LIN {X 0,Y 532.098,Z 319.802,A -85,B 0,C 180,E1 -4422.927,E2 -4422.927} C_VEL
LIN {X 0,Y 532.084,Z 308.331,A -85,B 0,C 180,E1 -4423.281,E2 -4423.281} C_VEL
LIN {X 0,Y 530.627,Z 298.644,A -85,B 0,C 180,E1 -4423.524,E2 -4423.524} C_VEL
LIN {X 0,Y 530.739,Z 289.457,A -85,B 0,C 180,E1 -4426.146,E2 -4426.146} C_VEL
LIN {X 0,Y 530.824,Z 279.726,A -85,B 0,C 180,E1 -4428.928,E2 -4428.928} C_VEL
LIN {X 0,Y 530.984,Z 268.988,A -85,B 0,C 180,E1 -4432.103,E2 -4432.103} C_VEL
LIN {X 0,Y 531.056,Z 259.338,A -85,B 0,C 180,E1 -4435.055,E2 -4435.055} C_VEL
LIN {X 0,Y 531.227,Z 250.169,A -85,B 0,C 180,E1 -4438.012,E2 -4438.012} C_VEL
LIN {X 0,Y 531.545,Z 241.433,A -85,B 0,C 180,E1 -4441.041,E2 -4441.041} C_VEL
LIN {X 0,Y 532.022,Z 233.376,A -85,B 0,C 180,E1 -4444.155,E2 -4444.155} C_VEL
LIN {X 0,Y 532.107,Z 230.247,A -85,B 0,C 180,E1 -4445.532,E2 -4445.532} C_VEL
LIN {X 0,Y 531.699,Z 226.333,A -85,B 0,C 180,E1 -4447.526,E2 -4447.526} C_VEL
LIN {X 0,Y 531.191,Z 223.293,A -85,B 0,C 180,E1 -4449.426,E2 -4449.426} C_VEL
LIN {X 0,Y 530.987,Z 222.375,A -85,B 0,C 180,E1 -4450.111,E2 -4450.111} C_VEL
LIN {X 0,Y 530.981,Z 222.346,A -85,B 0,C 180,E1 -4452.457,E2 -4452.457} C_VEL
LIN {X 0,Y 530.981,Z 222.348,A -85,B 0,C 180,E1 -4455.622,E2 -4455.622} C_VEL
LIN {X 0,Y 530.997,Z 222.344,A -85,B 0,C 180,E1 -4458.565,E2 -4458.565} C_VEL
LIN {X 0,Y 530.962,Z 222.35,A -85,B 0,C 180,E1 -4461.53,E2 -4461.53} C_VEL
LIN {X 0,Y 530.954,Z 222.351,A -85,B 0,C 180,E1 -4464.38,E2 -4464.38} C_VEL
LIN {X 0,Y 530.987,Z 222.799,A -85,B 0,C 180,E1 -4465.31,E2 -4465.31} C_VEL
LIN {X 0,Y 530.925,Z 225.158,A -85,B 0,C 180,E1 -4468.029,E2 -4468.029} C_VEL
LIN {X 0,Y 530.845,Z 227.83,A -85,B 0,C 180,E1 -4470.903,E2 -4470.903} C_VEL
LIN {X 0,Y 530.76,Z 231.038,A -85,B 0,C 180,E1 -4474.213,E2 -4474.213} C_VEL
LIN {X 0,Y 530.662,Z 233.419,A -85,B 0,C 180,E1 -4476.59,E2 -4476.59} C_VEL
LIN {X 0,Y 530.617,Z 235.93,A -85,B 0,C 180,E1 -4479.046,E2 -4479.046} C_VEL
LIN {X 0,Y 530.598,Z 239.55,A -85,B 0,C 180,E1 -4482.493,E2 -4482.493} C_VEL
LIN {X 0,Y 530.553,Z 242.668,A -85,B 0,C 180,E1 -4485.423,E2 -4485.423} C_VEL
LIN {X 0,Y 530.522,Z 245.123,A -85,B 0,C 180,E1 -4487.605,E2 -4487.605} C_VEL
LIN {X 0,Y 532.268,Z 254.517,A -85,B 0,C 180,E1 -4487.886,E2 -4487.886} C_VEL
LIN {X 0,Y 532.14,Z 267.138,A -85,B 0,C 180,E1 -4488.336,E2 -4488.336} C_VEL
LIN {X 0,Y 531.892,Z 278.037,A -85,B 0,C 180,E1 -4488.858,E2 -4488.858} C_VEL
LIN {X 0,Y 531.608,Z 288.977,A -85,B 0,C 180,E1 -4489.527,E2 -4489.527} C_VEL
LIN {X 0,Y 531.384,Z 300.143,A -85,B 0,C 180,E1 -4490.388,E2 -4490.388} C_VEL
LIN {X 0,Y 531.175,Z 309.139,A -85,B 0,C 180,E1 -4491.248,E2 -4491.248} C_VEL
LIN {X 0,Y 530.932,Z 317.38,A -85,B 0,C 180,E1 -4492.202,E2 -4492.202} C_VEL
LIN {X 0,Y 530.778,Z 324.845,A -85,B 0,C 180,E1 -4493.255,E2 -4493.255} C_VEL
LIN {X 0,Y 530.663,Z 330.911,A -85,B 0,C 180,E1 -4494.3,E2 -4494.3} C_VEL
LIN {X 0,Y 530.602,Z 336.255,A -85,B 0,C 180,E1 -4495.442,E2 -4495.442} C_VEL
LIN {X 0,Y 530.567,Z 340.431,A -85,B 0,C 180,E1 -4496.583,E2 -4496.583} C_VEL
LIN {X 0,Y 530.431,Z 343.565,A -85,B 0,C 180,E1 -4497.722,E2 -4497.722} C_VEL
LIN {X 0,Y 530.373,Z 345.123,A -85,B 0,C 180,E1 -4498.481,E2 -4498.481} C_VEL
LIN {X 0,Y 530.355,Z 346.27,A -85,B 0,C 180,E1 -4499.241,E2 -4499.241} C_VEL
LIN {X 0,Y 530.351,Z 347.32,A -85,B 0,C 180,E1 -4500.759,E2 -4500.759} C_VEL
LIN {X 0,Y 530.411,Z 346.844,A -85,B 0,C 180,E1 -4502.278,E2 -4502.278} C_VEL
LIN {X 0,Y 530.482,Z 345.982,A -85,B 0,C 180,E1 -4503.038,E2 -4503.038} C_VEL
LIN {X 0,Y 530.489,Z 344.731,A -85,B 0,C 180,E1 -4503.798,E2 -4503.798} C_VEL
LIN {X 0,Y 530.441,Z 342.081,A -85,B 0,C 180,E1 -4504.941,E2 -4504.941} C_VEL
LIN {X 0,Y 530.554,Z 338.414,A -85,B 0,C 180,E1 -4506.083,E2 -4506.083} C_VEL
LIN {X 0,Y 530.61,Z 333.633,A -85,B 0,C 180,E1 -4507.229,E2 -4507.229} C_VEL
LIN {X 0,Y 530.755,Z 327.585,A -85,B 0,C 180,E1 -4508.375,E2 -4508.375} C_VEL
LIN {X 0,Y 530.878,Z 320.048,A -85,B 0,C 180,E1 -4509.525,E2 -4509.525} C_VEL
LIN {X 0,Y 531.079,Z 312.325,A -85,B 0,C 180,E1 -4510.484,E2 -4510.484} C_VEL
LIN {X 0,Y 531.333,Z 302.877,A -85,B 0,C 180,E1 -4511.444,E2 -4511.444} C_VEL
LIN {X 0,Y 531.503,Z 292.376,A -85,B 0,C 180,E1 -4512.311,E2 -4512.311} C_VEL
LIN {X 0,Y 531.862,Z 280.673,A -85,B 0,C 180,E1 -4513.079,E2 -4513.079} C_VEL
LIN {X 0,Y 532.065,Z 268.141,A -85,B 0,C 180,E1 -4513.706,E2 -4513.706} C_VEL
LIN {X 0,Y 532.272,Z 254.968,A -85,B 0,C 180,E1 -4514.188,E2 -4514.188} C_VEL
LIN {X 0,Y 530.472,Z 244.548,A -85,B 0,C 180,E1 -4514.506,E2 -4514.506} C_VEL
LIN {X 0,Y 530.488,Z 240.752,A -85,B 0,C 180,E1 -4517.741,E2 -4517.741} C_VEL
LIN {X 0,Y 530.476,Z 237.972,A -85,B 0,C 180,E1 -4520.149,E2 -4520.149} C_VEL
LIN {X 0,Y 530.473,Z 235.149,A -85,B 0,C 180,E1 -4522.595,E2 -4522.595} C_VEL
LIN {X 0,Y 530.536,Z 232.305,A -85,B 0,C 180,E1 -4525.081,E2 -4525.081} C_VEL
LIN {X 0,Y 530.579,Z 229.376,A -85,B 0,C 180,E1 -4527.62,E2 -4527.62} C_VEL
LIN {X 0,Y 530.596,Z 226.016,A -85,B 0,C 180,E1 -4530.575,E2 -4530.575} C_VEL
LIN {X 0,Y 530.623,Z 222.811,A -85,B 0,C 180,E1 -4533.443,E2 -4533.443} C_VEL
LIN {X 0,Y 530.64,Z 222.412,A -85,B 0,C 180,E1 -4533.798,E2 -4533.798} C_VEL
LIN {X 0,Y 530.907,Z 222.354,A -85,B 0,C 180,E1 -4536.563,E2 -4536.563} C_VEL
LIN {X 0,Y 530.94,Z 222.347,A -85,B 0,C 180,E1 -4538.185,E2 -4538.185} C_VEL
LIN {X 0,Y 530.31,Z 222.429,A -85,B 0,C 180,E1 -4538.819,E2 -4538.819} C_VEL
LIN {X 0,Y 527.489,Z 222.782,A -85,B 0,C 180,E1 -4539.847,E2 -4539.847} C_VEL
LIN {X 0,Y 525.079,Z 223.08,A -85,B 0,C 180,E1 -4540.674,E2 -4540.674} C_VEL
LIN {X 0,Y 524.034,Z 223.208,A -85,B 0,C 180,E1 -4541.314,E2 -4541.314} C_VEL
LIN {X 0,Y 523.944,Z 223.219,A -85,B 0,C 180,E1 -4541.53,E2 -4541.53} C_VEL
LIN {X 0,Y 523.945,Z 223.217,A -85,B 0,C 180,E1 -4544.689,E2 -4544.689} C_VEL
LIN {X 0,Y 523.912,Z 223.222,A -85,B 0,C 180,E1 -4547.877,E2 -4547.877} C_VEL
LIN {X 0,Y 523.903,Z 223.228,A -85,B 0,C 180,E1 -4550.913,E2 -4550.913} C_VEL
LIN {X 0,Y 523.858,Z 223.227,A -85,B 0,C 180,E1 -4553.821,E2 -4553.821} C_VEL
LIN {X 0,Y 523.916,Z 223.227,A -85,B 0,C 180,E1 -4556.633,E2 -4556.633} C_VEL
LIN {X 0,Y 523.948,Z 223.216,A -85,B 0,C 180,E1 -4559.355,E2 -4559.355} C_VEL
LIN {X 0,Y 523.951,Z 223.221,A -85,B 0,C 180,E1 -4562.288,E2 -4562.288} C_VEL
LIN {X 0,Y 523.932,Z 223.22,A -85,B 0,C 180,E1 -4564.58,E2 -4564.58} C_VEL
LIN {X 0,Y 523.915,Z 223.223,A -85,B 0,C 180,E1 -4567.106,E2 -4567.106} C_VEL
LIN {X 0,Y 523.984,Z 223.215,A -85,B 0,C 180,E1 -4569.866,E2 -4569.866} C_VEL
LIN {X 0,Y 523.955,Z 223.22,A -85,B 0,C 180,E1 -4572.837,E2 -4572.837} C_VEL
LIN {X 0,Y 523.978,Z 223.218,A -85,B 0,C 180,E1 -4575.236,E2 -4575.236} C_VEL
LIN {X 0,Y 524.018,Z 223.213,A -85,B 0,C 180,E1 -4578.394,E2 -4578.394} C_VEL
LIN {X 0,Y 523.957,Z 223.216,A -85,B 0,C 180,E1 -4581.515,E2 -4581.515} C_VEL
LIN {X 0,Y 524.028,Z 223.208,A -85,B 0,C 180,E1 -4584.613,E2 -4584.613} C_VEL
LIN {X 0,Y 524.106,Z 223.202,A -85,B 0,C 180,E1 -4587.694,E2 -4587.694} C_VEL
LIN {X 0,Y 524.104,Z 223.2,A -85,B 0,C 180,E1 -4590,E2 -4590} C_VEL
LIN {X 0,Y 524.043,Z 223.208,A -85,B 0,C 180,E1 -4593.075,E2 -4593.075} C_VEL
LIN {X 0,Y 523.728,Z 223.269,A -85,B 0,C 180,E1 -4595.728,E2 -4595.728} C_VEL
LIN {X 0,Y 523.74,Z 227.795,A -85,B 0,C 180,E1 -4597.712,E2 -4597.712} C_VEL
LIN {X 0,Y 523.7,Z 234.811,A -85,B 0,C 180,E1 -4600.829,E2 -4600.829} C_VEL
LIN {X 0,Y 523.643,Z 241.835,A -85,B 0,C 180,E1 -4603.98,E2 -4603.98} C_VEL
LIN {X 0,Y 523.592,Z 247.093,A -85,B 0,C 180,E1 -4606.372,E2 -4606.372} C_VEL
LIN {X 0,Y 523.568,Z 252.374,A -85,B 0,C 180,E1 -4608.793,E2 -4608.793} C_VEL
LIN {X 0,Y 523.481,Z 257.718,A -85,B 0,C 180,E1 -4611.253,E2 -4611.253} C_VEL
LIN {X 0,Y 523.449,Z 263.864,A -85,B 0,C 180,E1 -4614.077,E2 -4614.077} C_VEL
LIN {X 0,Y 523.466,Z 268.522,A -85,B 0,C 180,E1 -4616.266,E2 -4616.266} C_VEL
LIN {X 0,Y 524.612,Z 277.602,A -85,B 0,C 180,E1 -4616.558,E2 -4616.558} C_VEL
LIN {X 0,Y 524.443,Z 289.493,A -85,B 0,C 180,E1 -4617.052,E2 -4617.052} C_VEL
LIN {X 0,Y 524.275,Z 298.999,A -85,B 0,C 180,E1 -4617.602,E2 -4617.602} C_VEL
LIN {X 0,Y 524.117,Z 307.314,A -85,B 0,C 180,E1 -4618.208,E2 -4618.208} C_VEL
LIN {X 0,Y 523.983,Z 314.738,A -85,B 0,C 180,E1 -4618.872,E2 -4618.872} C_VEL
LIN {X 0,Y 523.833,Z 321.728,A -85,B 0,C 180,E1 -4619.631,E2 -4619.631} C_VEL
LIN {X 0,Y 523.656,Z 329.312,A -85,B 0,C 180,E1 -4620.664,E2 -4620.664} C_VEL
LIN {X 0,Y 523.583,Z 334.586,A -85,B 0,C 180,E1 -4621.567,E2 -4621.567} C_VEL
LIN {X 0,Y 523.433,Z 338.885,A -85,B 0,C 180,E1 -4622.484,E2 -4622.484} C_VEL
LIN {X 0,Y 523.417,Z 343.011,A -85,B 0,C 180,E1 -4623.645,E2 -4623.645} C_VEL
LIN {X 0,Y 523.316,Z 346.207,A -85,B 0,C 180,E1 -4624.993,E2 -4624.993} C_VEL
LIN {X 0,Y 523.293,Z 347.688,A -85,B 0,C 180,E1 -4626.31,E2 -4626.31} C_VEL
LIN {X 0,Y 523.248,Z 347.784,A -85,B 0,C 180,E1 -4627.584,E2 -4627.584} C_VEL
LIN {X 0,Y 523.269,Z 347.456,A -85,B 0,C 180,E1 -4628.158,E2 -4628.158} C_VEL
LIN {X 0,Y 523.312,Z 346.143,A -85,B 0,C 180,E1 -4629.139,E2 -4629.139} C_VEL
LIN {X 0,Y 523.389,Z 343.95,A -85,B 0,C 180,E1 -4630.131,E2 -4630.131} C_VEL
LIN {X 0,Y 523.435,Z 340.367,A -85,B 0,C 180,E1 -4631.245,E2 -4631.245} C_VEL
LIN {X 0,Y 523.516,Z 335.247,A -85,B 0,C 180,E1 -4632.408,E2 -4632.408} C_VEL
LIN {X 0,Y 523.624,Z 329.683,A -85,B 0,C 180,E1 -4633.378,E2 -4633.378} C_VEL
LIN {X 0,Y 523.771,Z 323.495,A -85,B 0,C 180,E1 -4634.246,E2 -4634.246} C_VEL
LIN {X 0,Y 523.966,Z 315.668,A -85,B 0,C 180,E1 -4635.132,E2 -4635.132} C_VEL
LIN {X 0,Y 524.107,Z 307.523,A -85,B 0,C 180,E1 -4635.871,E2 -4635.871} C_VEL
LIN {X 0,Y 524.296,Z 298.844,A -85,B 0,C 180,E1 -4636.504,E2 -4636.504} C_VEL
LIN {X 0,Y 524.511,Z 288.092,A -85,B 0,C 180,E1 -4637.111,E2 -4637.111} C_VEL
LIN {X 0,Y 524.614,Z 276.997,A -85,B 0,C 180,E1 -4637.554,E2 -4637.554} C_VEL
LIN {X 0,Y 523.439,Z 268.659,A -85,B 0,C 180,E1 -4637.83,E2 -4637.83} C_VEL
LIN {X 0,Y 523.494,Z 262.077,A -85,B 0,C 180,E1 -4640.877,E2 -4640.877} C_VEL
LIN {X 0,Y 523.487,Z 255.721,A -85,B 0,C 180,E1 -4643.792,E2 -4643.792} C_VEL
LIN {X 0,Y 523.611,Z 249.505,A -85,B 0,C 180,E1 -4646.611,E2 -4646.611} C_VEL
LIN {X 0,Y 523.578,Z 243.42,A -85,B 0,C 180,E1 -4649.331,E2 -4649.331} C_VEL
LIN {X 0,Y 523.635,Z 237.419,A -85,B 0,C 180,E1 -4651.981,E2 -4651.981} C_VEL
LIN {X 0,Y 523.641,Z 230.395,A -85,B 0,C 180,E1 -4654.99,E2 -4654.99} C_VEL
LIN {X 0,Y 523.728,Z 223.254,A -85,B 0,C 180,E1 -4657.982,E2 -4657.982} C_VEL
LIN {X 0,Y 523.963,Z 223.22,A -85,B 0,C 180,E1 -4660.407,E2 -4660.407} C_VEL
LIN {X 0,Y 523.958,Z 223.22,A -85,B 0,C 180,E1 -4662.837,E2 -4662.837} C_VEL
LIN {X 0,Y 523.979,Z 223.217,A -85,B 0,C 180,E1 -4665.236,E2 -4665.236} C_VEL
LIN {X 0,Y 524.016,Z 223.215,A -85,B 0,C 180,E1 -4668.394,E2 -4668.394} C_VEL
LIN {X 0,Y 524.007,Z 223.214,A -85,B 0,C 180,E1 -4671.516,E2 -4671.516} C_VEL
LIN {X 0,Y 524.075,Z 223.205,A -85,B 0,C 180,E1 -4674.613,E2 -4674.613} C_VEL
LIN {X 0,Y 524.115,Z 223.202,A -85,B 0,C 180,E1 -4677.694,E2 -4677.694} C_VEL
LIN {X 0,Y 524.124,Z 223.199,A -85,B 0,C 180,E1 -4680.768,E2 -4680.768} C_VEL
LIN {X 0,Y 524.072,Z 223.205,A -85,B 0,C 180,E1 -4683.075,E2 -4683.075} C_VEL
LIN {X 0,Y 524.029,Z 223.213,A -85,B 0,C 180,E1 -4686.159,E2 -4686.159} C_VEL
LIN {X 0,Y 524.004,Z 223.216,A -85,B 0,C 180,E1 -4688.484,E2 -4688.484} C_VEL
LIN {X 0,Y 524.007,Z 223.214,A -85,B 0,C 180,E1 -4691.739,E2 -4691.739} C_VEL
LIN {X 0,Y 523.997,Z 223.215,A -85,B 0,C 180,E1 -4695.052,E2 -4695.052} C_VEL
LIN {X 0,Y 523.95,Z 223.223,A -85,B 0,C 180,E1 -4697.969,E2 -4697.969} C_VEL
LIN {X 0,Y 523.975,Z 223.219,A -85,B 0,C 180,E1 -4700.41,E2 -4700.41} C_VEL
LIN {X 0,Y 523.914,Z 223.227,A -85,B 0,C 180,E1 -4702.893,E2 -4702.893} C_VEL
LIN {X 0,Y 523.946,Z 223.222,A -85,B 0,C 180,E1 -4706.01,E2 -4706.01} C_VEL
LIN {X 0,Y 523.937,Z 223.222,A -85,B 0,C 180,E1 -4708.875,E2 -4708.875} C_VEL
LIN {X 0,Y 523.922,Z 223.223,A -85,B 0,C 180,E1 -4711.544,E2 -4711.544} C_VEL
LIN {X 0,Y 523.923,Z 223.224,A -85,B 0,C 180,E1 -4714.291,E2 -4714.291} C_VEL
LIN {X 0,Y 523.91,Z 223.227,A -85,B 0,C 180,E1 -4717.132,E2 -4717.132} C_VEL
LIN {X 0,Y 523.94,Z 223.221,A -85,B 0,C 180,E1 -4720.13,E2 -4720.13} C_VEL
LIN {X 0,Y 523.937,Z 223.222,A -85,B 0,C 180,E1 -4722.459,E2 -4722.459} C_VEL
LIN {X 0,Y 523.946,Z 223.224,A -85,B 0,C 180,E1 -4725.31,E2 -4725.31} C_VEL
LIN {X 0,Y 523.958,Z 223.221,A -85,B 0,C 180,E1 -4728.69,E2 -4728.69} C_VEL
LIN {X 0,Y 523.954,Z 223.362,A -85,B 0,C 180,E1 -4731.595,E2 -4731.595} C_VEL
LIN {X 0,Y 524.95,Z 229.317,A -85,B 0,C 180,E1 -4733.909,E2 -4733.909} C_VEL
LIN {X 0,Y 524.989,Z 235.318,A -85,B 0,C 180,E1 -4736.098,E2 -4736.098} C_VEL
LIN {X 0,Y 524.695,Z 243.654,A -85,B 0,C 180,E1 -4739.009,E2 -4739.009} C_VEL
LIN {X 0,Y 524.336,Z 253.187,A -85,B 0,C 180,E1 -4742.207,E2 -4742.207} C_VEL
LIN {X 0,Y 524.169,Z 261.804,A -85,B 0,C 180,E1 -4745.017,E2 -4745.017} C_VEL
LIN {X 0,Y 523.984,Z 271.06,A -85,B 0,C 180,E1 -4747.941,E2 -4747.941} C_VEL
LIN {X 0,Y 523.837,Z 280.341,A -85,B 0,C 180,E1 -4750.81,E2 -4750.81} C_VEL
LIN {X 0,Y 523.672,Z 291.052,A -85,B 0,C 180,E1 -4754.031,E2 -4754.031} C_VEL
LIN {X 0,Y 523.592,Z 298.662,A -85,B 0,C 180,E1 -4756.291,E2 -4756.291} C_VEL
LIN {X 0,Y 525.346,Z 311.496,A -85,B 0,C 180,E1 -4756.633,E2 -4756.633} C_VEL
LIN {X 0,Y 525.105,Z 323.517,A -85,B 0,C 180,E1 -4757.045,E2 -4757.045} C_VEL
LIN {X 0,Y 524.816,Z 335.824,A -85,B 0,C 180,E1 -4757.628,E2 -4757.628} C_VEL
LIN {X 0,Y 524.526,Z 346.977,A -85,B 0,C 180,E1 -4758.31,E2 -4758.31} C_VEL
LIN {X 0,Y 524.308,Z 358.307,A -85,B 0,C 180,E1 -4759.184,E2 -4759.184} C_VEL
LIN {X 0,Y 524.003,Z 368.366,A -85,B 0,C 180,E1 -4760.154,E2 -4760.154} C_VEL
LIN {X 0,Y 523.776,Z 378.119,A -85,B 0,C 180,E1 -4761.318,E2 -4761.318} C_VEL
LIN {X 0,Y 523.612,Z 385.896,A -85,B 0,C 180,E1 -4762.48,E2 -4762.48} C_VEL
LIN {X 0,Y 523.482,Z 393.051,A -85,B 0,C 180,E1 -4763.834,E2 -4763.834} C_VEL
LIN {X 0,Y 523.383,Z 397.812,A -85,B 0,C 180,E1 -4764.993,E2 -4764.993} C_VEL
LIN {X 0,Y 523.443,Z 401.456,A -85,B 0,C 180,E1 -4766.151,E2 -4766.151} C_VEL
LIN {X 0,Y 523.367,Z 403.328,A -85,B 0,C 180,E1 -4766.921,E2 -4766.921} C_VEL
LIN {X 0,Y 523.335,Z 404.733,A -85,B 0,C 180,E1 -4767.691,E2 -4767.691} C_VEL
LIN {X 0,Y 523.254,Z 406.343,A -85,B 0,C 180,E1 -4769.231,E2 -4769.231} C_VEL
LIN {X 0,Y 523.254,Z 406.556,A -85,B 0,C 180,E1 -4770,E2 -4770} C_VEL
LIN {X 0,Y 523.275,Z 405.721,A -85,B 0,C 180,E1 -4771.539,E2 -4771.539} C_VEL
LIN {X 0,Y 523.335,Z 404.718,A -85,B 0,C 180,E1 -4772.309,E2 -4772.309} C_VEL
LIN {X 0,Y 523.367,Z 403.301,A -85,B 0,C 180,E1 -4773.079,E2 -4773.079} C_VEL
LIN {X 0,Y 523.424,Z 400.331,A -85,B 0,C 180,E1 -4774.235,E2 -4774.235} C_VEL
LIN {X 0,Y 523.461,Z 396.306,A -85,B 0,C 180,E1 -4775.393,E2 -4775.393} C_VEL
LIN {X 0,Y 523.515,Z 391.014,A -85,B 0,C 180,E1 -4776.574,E2 -4776.574} C_VEL
LIN {X 0,Y 523.649,Z 384.588,A -85,B 0,C 180,E1 -4777.713,E2 -4777.713} C_VEL
LIN {X 0,Y 523.821,Z 376.445,A -85,B 0,C 180,E1 -4778.876,E2 -4778.876} C_VEL
LIN {X 0,Y 523.992,Z 368.138,A -85,B 0,C 180,E1 -4779.847,E2 -4779.847} C_VEL
LIN {X 0,Y 524.267,Z 358.003,A -85,B 0,C 180,E1 -4780.817,E2 -4780.817} C_VEL
LIN {X 0,Y 524.475,Z 347.981,A -85,B 0,C 180,E1 -4781.596,E2 -4781.596} C_VEL
LIN {X 0,Y 524.734,Z 336.619,A -85,B 0,C 180,E1 -4782.304,E2 -4782.304} C_VEL
LIN {X 0,Y 525.055,Z 324.104,A -85,B 0,C 180,E1 -4782.907,E2 -4782.907} C_VEL
LIN {X 0,Y 525.275,Z 311.692,A -85,B 0,C 180,E1 -4783.344,E2 -4783.344} C_VEL
LIN {X 0,Y 523.553,Z 298.144,A -85,B 0,C 180,E1 -4783.71,E2 -4783.71} C_VEL
LIN {X 0,Y 523.67,Z 287.615,A -85,B 0,C 180,E1 -4786.771,E2 -4786.771} C_VEL
LIN {X 0,Y 523.757,Z 277.96,A -85,B 0,C 180,E1 -4789.601,E2 -4789.601} C_VEL
LIN {X 0,Y 523.908,Z 268.267,A -85,B 0,C 180,E1 -4792.527,E2 -4792.527} C_VEL
LIN {X 0,Y 524.023,Z 259.064,A -85,B 0,C 180,E1 -4795.415,E2 -4795.415} C_VEL
LIN {X 0,Y 524.202,Z 250.009,A -85,B 0,C 180,E1 -4798.422,E2 -4798.422} C_VEL
LIN {X 0,Y 524.518,Z 242.878,A -85,B 0,C 180,E1 -4800.959,E2 -4800.959} C_VEL
LIN {X 0,Y 524.985,Z 235.381,A -85,B 0,C 180,E1 -4803.901,E2 -4803.901} C_VEL
LIN {X 0,Y 525.146,Z 232.248,A -85,B 0,C 180,E1 -4805.278,E2 -4805.278} C_VEL
LIN {X 0,Y 524.87,Z 228.733,A -85,B 0,C 180,E1 -4807.053,E2 -4807.053} C_VEL
LIN {X 0,Y 524.387,Z 225.445,A -85,B 0,C 180,E1 -4809.044,E2 -4809.044} C_VEL
LIN {X 0,Y 524.087,Z 223.945,A -85,B 0,C 180,E1 -4810.149,E2 -4810.149} C_VEL
LIN {X 0,Y 523.959,Z 223.223,A -85,B 0,C 180,E1 -4811.31,E2 -4811.31} C_VEL
LIN {X 0,Y 523.947,Z 223.222,A -85,B 0,C 180,E1 -4814.69,E2 -4814.69} C_VEL
LIN {X 0,Y 523.955,Z 223.223,A -85,B 0,C 180,E1 -4817.881,E2 -4817.881} C_VEL
LIN {X 0,Y 523.924,Z 223.226,A -85,B 0,C 180,E1 -4820.915,E2 -4820.915} C_VEL
LIN {X 0,Y 523.903,Z 223.229,A -85,B 0,C 180,E1 -4823.825,E2 -4823.825} C_VEL
LIN {X 0,Y 523.955,Z 223.576,A -85,B 0,C 180,E1 -4824.907,E2 -4824.907} C_VEL
LIN {X 0,Y 523.907,Z 225.869,A -85,B 0,C 180,E1 -4827.686,E2 -4827.686} C_VEL
LIN {X 0,Y 523.805,Z 228.57,A -85,B 0,C 180,E1 -4830.707,E2 -4830.707} C_VEL
LIN {X 0,Y 523.695,Z 231.404,A -85,B 0,C 180,E1 -4833.713,E2 -4833.713} C_VEL
LIN {X 0,Y 523.64,Z 233.9,A -85,B 0,C 180,E1 -4836.256,E2 -4836.256} C_VEL
LIN {X 0,Y 523.559,Z 236.392,A -85,B 0,C 180,E1 -4838.75,E2 -4838.75} C_VEL
LIN {X 0,Y 523.504,Z 238.935,A -85,B 0,C 180,E1 -4841.204,E2 -4841.204} C_VEL
LIN {X 0,Y 523.481,Z 241.49,A -85,B 0,C 180,E1 -4843.624,E2 -4843.624} C_VEL
LIN {X 0,Y 523.457,Z 244.046,A -85,B 0,C 180,E1 -4846.015,E2 -4846.015} C_VEL
LIN {X 0,Y 523.445,Z 245.666,A -85,B 0,C 180,E1 -4847.429,E2 -4847.429} C_VEL
LIN {X 0,Y 525.349,Z 255.262,A -85,B 0,C 180,E1 -4847.727,E2 -4847.727} C_VEL
LIN {X 0,Y 525.202,Z 267.853,A -85,B 0,C 180,E1 -4848.188,E2 -4848.188} C_VEL
LIN {X 0,Y 524.921,Z 280.258,A -85,B 0,C 180,E1 -4848.806,E2 -4848.806} C_VEL
LIN {X 0,Y 524.608,Z 290.84,A -85,B 0,C 180,E1 -4849.483,E2 -4849.483} C_VEL
LIN {X 0,Y 524.37,Z 301.659,A -85,B 0,C 180,E1 -4850.356,E2 -4850.356} C_VEL
LIN {X 0,Y 524.14,Z 311.352,A -85,B 0,C 180,E1 -4851.324,E2 -4851.324} C_VEL
LIN {X 0,Y 523.892,Z 319.298,A -85,B 0,C 180,E1 -4852.291,E2 -4852.291} C_VEL
LIN {X 0,Y 523.741,Z 327.294,A -85,B 0,C 180,E1 -4853.487,E2 -4853.487} C_VEL
LIN {X 0,Y 523.502,Z 333.296,A -85,B 0,C 180,E1 -4854.608,E2 -4854.608} C_VEL
LIN {X 0,Y 523.496,Z 338.221,A -85,B 0,C 180,E1 -4855.766,E2 -4855.766} C_VEL
LIN {X 0,Y 523.475,Z 342.031,A -85,B 0,C 180,E1 -4856.922,E2 -4856.922} C_VEL
LIN {X 0,Y 523.356,Z 343.998,A -85,B 0,C 180,E1 -4857.691,E2 -4857.691} C_VEL
LIN {X 0,Y 523.289,Z 345.551,A -85,B 0,C 180,E1 -4858.461,E2 -4858.461} C_VEL
LIN {X 0,Y 523.269,Z 346.69,A -85,B 0,C 180,E1 -4859.231,E2 -4859.231} C_VEL
LIN {X 0,Y 523.263,Z 347.725,A -85,B 0,C 180,E1 -4860.77,E2 -4860.77} C_VEL
LIN {X 0,Y 523.335,Z 347.223,A -85,B 0,C 180,E1 -4862.309,E2 -4862.309} C_VEL
LIN {X 0,Y 523.418,Z 346.347,A -85,B 0,C 180,E1 -4863.079,E2 -4863.079} C_VEL
LIN {X 0,Y 523.411,Z 345.086,A -85,B 0,C 180,E1 -4863.85,E2 -4863.85} C_VEL
LIN {X 0,Y 523.367,Z 342.41,A -85,B 0,C 180,E1 -4865.008,E2 -4865.008} C_VEL
LIN {X 0,Y 523.494,Z 338.714,A -85,B 0,C 180,E1 -4866.166,E2 -4866.166} C_VEL
LIN {X 0,Y 523.552,Z 333.901,A -85,B 0,C 180,E1 -4867.327,E2 -4867.327} C_VEL
LIN {X 0,Y 523.722,Z 327.816,A -85,B 0,C 180,E1 -4868.489,E2 -4868.489} C_VEL
LIN {X 0,Y 523.853,Z 320.233,A -85,B 0,C 180,E1 -4869.654,E2 -4869.654} C_VEL
LIN {X 0,Y 524.082,Z 312.46,A -85,B 0,C 180,E1 -4870.626,E2 -4870.626} C_VEL
LIN {X 0,Y 524.332,Z 302.953,A -85,B 0,C 180,E1 -4871.599,E2 -4871.599} C_VEL
LIN {X 0,Y 524.538,Z 292.395,A -85,B 0,C 180,E1 -4872.477,E2 -4872.477} C_VEL
LIN {X 0,Y 524.917,Z 280.59,A -85,B 0,C 180,E1 -4873.255,E2 -4873.255} C_VEL
LIN {X 0,Y 525.128,Z 267.944,A -85,B 0,C 180,E1 -4873.891,E2 -4873.891} C_VEL
LIN {X 0,Y 525.325,Z 255.019,A -85,B 0,C 180,E1 -4874.367,E2 -4874.367} C_VEL
LIN {X 0,Y 523.424,Z 244.888,A -85,B 0,C 180,E1 -4874.694,E2 -4874.694} C_VEL
LIN {X 0,Y 523.393,Z 241.047,A -85,B 0,C 180,E1 -4877.989,E2 -4877.989} C_VEL
LIN {X 0,Y 523.391,Z 238.196,A -85,B 0,C 180,E1 -4880.434,E2 -4880.434} C_VEL
LIN {X 0,Y 523.401,Z 235.35,A -85,B 0,C 180,E1 -4882.917,E2 -4882.917} C_VEL
LIN {X 0,Y 523.531,Z 231.923,A -85,B 0,C 180,E1 -4885.917,E2 -4885.917} C_VEL
LIN {X 0,Y 523.495,Z 228.52,A -85,B 0,C 180,E1 -4888.902,E2 -4888.902} C_VEL
LIN {X 0,Y 523.546,Z 225.542,A -85,B 0,C 180,E1 -4891.57,E2 -4891.57} C_VEL
LIN {X 0,Y 523.581,Z 223.27,A -85,B 0,C 180,E1 -4893.671,E2 -4893.671} C_VEL
LIN {X 0,Y 523.849,Z 223.234,A -85,B 0,C 180,E1 -4896.393,E2 -4896.393} C_VEL
LIN {X 0,Y 523.925,Z 223.22,A -85,B 0,C 180,E1 -4899.085,E2 -4899.085} C_VEL
LIN {X 0,Y 523.944,Z 223.219,A -85,B 0,C 180,E1 -4901.53,E2 -4901.53} C_VEL
LIN {X 0,Y 523.256,Z 223.306,A -85,B 0,C 180,E1 -4902.171,E2 -4902.171} C_VEL
LIN {X 0,Y 520.369,Z 223.665,A -85,B 0,C 180,E1 -4903.211,E2 -4903.211} C_VEL
LIN {X 0,Y 517.959,Z 223.966,A -85,B 0,C 180,E1 -4904.049,E2 -4904.049} C_VEL
LIN {X 0,Y 516.957,Z 224.088,A -85,B 0,C 180,E1 -4904.697,E2 -4904.697} C_VEL
LIN {X 0,Y 516.892,Z 224.097,A -85,B 0,C 180,E1 -4904.916,E2 -4904.916} C_VEL
LIN {X 0,Y 516.887,Z 224.096,A -85,B 0,C 180,E1 -4908.222,E2 -4908.222} C_VEL
LIN {X 0,Y 516.865,Z 224.102,A -85,B 0,C 180,E1 -4911.282,E2 -4911.282} C_VEL
LIN {X 0,Y 516.852,Z 224.107,A -85,B 0,C 180,E1 -4914.673,E2 -4914.673} C_VEL
LIN {X 0,Y 516.897,Z 224.094,A -85,B 0,C 180,E1 -4917.457,E2 -4917.457} C_VEL
LIN {X 0,Y 516.924,Z 224.094,A -85,B 0,C 180,E1 -4920.695,E2 -4920.695} C_VEL
LIN {X 0,Y 516.915,Z 224.098,A -85,B 0,C 180,E1 -4923.811,E2 -4923.811} C_VEL
LIN {X 0,Y 516.865,Z 224.1,A -85,B 0,C 180,E1 -4926.776,E2 -4926.776} C_VEL
LIN {X 0,Y 516.944,Z 224.094,A -85,B 0,C 180,E1 -4929.732,E2 -4929.732} C_VEL
LIN {X 0,Y 516.908,Z 224.096,A -85,B 0,C 180,E1 -4932.595,E2 -4932.595} C_VEL
LIN {X 0,Y 516.944,Z 224.094,A -85,B 0,C 180,E1 -4935.03,E2 -4935.03} C_VEL
LIN {X 0,Y 516.971,Z 224.089,A -85,B 0,C 180,E1 -4938.234,E2 -4938.234} C_VEL
LIN {X 0,Y 516.933,Z 224.091,A -85,B 0,C 180,E1 -4941.399,E2 -4941.399} C_VEL
LIN {X 0,Y 516.979,Z 224.087,A -85,B 0,C 180,E1 -4944.539,E2 -4944.539} C_VEL
LIN {X 0,Y 517.076,Z 224.077,A -85,B 0,C 180,E1 -4947.663,E2 -4947.663} C_VEL
LIN {X 0,Y 517.073,Z 224.076,A -85,B 0,C 180,E1 -4950,E2 -4950} C_VEL
LIN {X 0,Y 517.084,Z 224.071,A -85,B 0,C 180,E1 -4952.337,E2 -4952.337} C_VEL
LIN {X 0,Y 516.8,Z 224.116,A -85,B 0,C 180,E1 -4955.462,E2 -4955.462} C_VEL
LIN {X 0,Y 516.693,Z 224.356,A -85,B 0,C 180,E1 -4955.855,E2 -4955.855} C_VEL
LIN {X 0,Y 516.663,Z 228.793,A -85,B 0,C 180,E1 -4957.818,E2 -4957.818} C_VEL
LIN {X 0,Y 516.635,Z 235.877,A -85,B 0,C 180,E1 -4960.979,E2 -4960.979} C_VEL
LIN {X 0,Y 516.578,Z 241.221,A -85,B 0,C 180,E1 -4963.373,E2 -4963.373} C_VEL
LIN {X 0,Y 516.549,Z 246.522,A -85,B 0,C 180,E1 -4965.79,E2 -4965.79} C_VEL
LIN {X 0,Y 516.504,Z 251.858,A -85,B 0,C 180,E1 -4968.238,E2 -4968.238} C_VEL
LIN {X 0,Y 516.424,Z 257.231,A -85,B 0,C 180,E1 -4970.722,E2 -4970.722} C_VEL
LIN {X 0,Y 516.411,Z 262.676,A -85,B 0,C 180,E1 -4973.245,E2 -4973.245} C_VEL
LIN {X 0,Y 516.387,Z 268.919,A -85,B 0,C 180,E1 -4976.128,E2 -4976.128} C_VEL
LIN {X 0,Y 517.649,Z 278.128,A -85,B 0,C 180,E1 -4976.424,E2 -4976.424} C_VEL
LIN {X 0,Y 517.467,Z 289.529,A -85,B 0,C 180,E1 -4976.9,E2 -4976.9} C_VEL
LIN {X 0,Y 517.27,Z 299.908,A -85,B 0,C 180,E1 -4977.513,E2 -4977.513} C_VEL
LIN {X 0,Y 517.093,Z 308.288,A -85,B 0,C 180,E1 -4978.141,E2 -4978.141} C_VEL
LIN {X 0,Y 516.946,Z 316.043,A -85,B 0,C 180,E1 -4978.857,E2 -4978.857} C_VEL
LIN {X 0,Y 516.795,Z 322.856,A -85,B 0,C 180,E1 -4979.626,E2 -4979.626} C_VEL
LIN {X 0,Y 516.625,Z 329.879,A -85,B 0,C 180,E1 -4980.606,E2 -4980.606} C_VEL
LIN {X 0,Y 516.503,Z 335.491,A -85,B 0,C 180,E1 -4981.592,E2 -4981.592} C_VEL
LIN {X 0,Y 516.359,Z 340.319,A -85,B 0,C 180,E1 -4982.687,E2 -4982.687} C_VEL
LIN {X 0,Y 516.335,Z 344.311,A -85,B 0,C 180,E1 -4983.922,E2 -4983.922} C_VEL
LIN {X 0,Y 516.207,Z 346.962,A -85,B 0,C 180,E1 -4985.226,E2 -4985.226} C_VEL
LIN {X 0,Y 516.209,Z 347.724,A -85,B 0,C 180,E1 -4985.833,E2 -4985.833} C_VEL
LIN {X 0,Y 516.19,Z 348.287,A -85,B 0,C 180,E1 -4986.803,E2 -4986.803} C_VEL
LIN {X 0,Y 516.168,Z 348.064,A -85,B 0,C 180,E1 -4987.841,E2 -4987.841} C_VEL
LIN {X 0,Y 516.243,Z 346.638,A -85,B 0,C 180,E1 -4989.105,E2 -4989.105} C_VEL
LIN {X 0,Y 516.325,Z 343.86,A -85,B 0,C 180,E1 -4990.337,E2 -4990.337} C_VEL
LIN {X 0,Y 516.392,Z 339.86,A -85,B 0,C 180,E1 -4991.535,E2 -4991.535} C_VEL
LIN {X 0,Y 516.497,Z 334.44,A -85,B 0,C 180,E1 -4992.711,E2 -4992.711} C_VEL
LIN {X 0,Y 516.639,Z 329.113,A -85,B 0,C 180,E1 -4993.613,E2 -4993.613} C_VEL
LIN {X 0,Y 516.789,Z 321.875,A -85,B 0,C 180,E1 -4994.593,E2 -4994.593} C_VEL
LIN {X 0,Y 517.016,Z 313.139,A -85,B 0,C 180,E1 -4995.533,E2 -4995.533} C_VEL
LIN {X 0,Y 517.234,Z 304.069,A -85,B 0,C 180,E1 -4996.294,E2 -4996.294} C_VEL
LIN {X 0,Y 517.377,Z 295.4,A -85,B 0,C 180,E1 -4996.869,E2 -4996.869} C_VEL
LIN {X 0,Y 517.556,Z 285.682,A -85,B 0,C 180,E1 -4997.37,E2 -4997.37} C_VEL
LIN {X 0,Y 517.572,Z 276.252,A -85,B 0,C 180,E1 -4997.734,E2 -4997.734} C_VEL
LIN {X 0,Y 516.383,Z 269.045,A -85,B 0,C 180,E1 -4997.975,E2 -4997.975} C_VEL
LIN {X 0,Y 516.443,Z 262.779,A -85,B 0,C 180,E1 -5000.867,E2 -5000.867} C_VEL
LIN {X 0,Y 516.424,Z 257.263,A -85,B 0,C 180,E1 -5003.411,E2 -5003.411} C_VEL
LIN {X 0,Y 516.543,Z 250.198,A -85,B 0,C 180,E1 -5006.566,E2 -5006.566} C_VEL
LIN {X 0,Y 516.526,Z 244.81,A -85,B 0,C 180,E1 -5009.004,E2 -5009.004} C_VEL
LIN {X 0,Y 516.574,Z 237.728,A -85,B 0,C 180,E1 -5012.169,E2 -5012.169} C_VEL
LIN {X 0,Y 516.59,Z 230.999,A -85,B 0,C 180,E1 -5015.055,E2 -5015.055} C_VEL
LIN {X 0,Y 516.661,Z 224.134,A -85,B 0,C 180,E1 -5017.945,E2 -5017.945} C_VEL
LIN {X 0,Y 516.92,Z 224.098,A -85,B 0,C 180,E1 -5020.129,E2 -5020.129} C_VEL
LIN {X 0,Y 516.909,Z 224.099,A -85,B 0,C 180,E1 -5022.595,E2 -5022.595} C_VEL
LIN {X 0,Y 516.945,Z 224.094,A -85,B 0,C 180,E1 -5025.03,E2 -5025.03} C_VEL
LIN {X 0,Y 516.969,Z 224.094,A -85,B 0,C 180,E1 -5028.234,E2 -5028.234} C_VEL
LIN {X 0,Y 516.972,Z 224.09,A -85,B 0,C 180,E1 -5031.4,E2 -5031.4} C_VEL
LIN {X 0,Y 517.02,Z 224.084,A -85,B 0,C 180,E1 -5034.54,E2 -5034.54} C_VEL
LIN {X 0,Y 517.087,Z 224.078,A -85,B 0,C 180,E1 -5037.663,E2 -5037.663} C_VEL
LIN {X 0,Y 517.095,Z 224.075,A -85,B 0,C 180,E1 -5040.779,E2 -5040.779} C_VEL
LIN {X 0,Y 517.013,Z 224.085,A -85,B 0,C 180,E1 -5043.117,E2 -5043.117} C_VEL
LIN {X 0,Y 516.992,Z 224.089,A -85,B 0,C 180,E1 -5046.243,E2 -5046.243} C_VEL
LIN {X 0,Y 516.969,Z 224.092,A -85,B 0,C 180,E1 -5048.6,E2 -5048.6} C_VEL
LIN {X 0,Y 516.956,Z 224.093,A -85,B 0,C 180,E1 -5051.807,E2 -5051.807} C_VEL
LIN {X 0,Y 516.948,Z 224.093,A -85,B 0,C 180,E1 -5055.146,E2 -5055.146} C_VEL
LIN {X 0,Y 516.919,Z 224.096,A -85,B 0,C 180,E1 -5058.222,E2 -5058.222} C_VEL
LIN {X 0,Y 516.915,Z 224.097,A -85,B 0,C 180,E1 -5060.701,E2 -5060.701} C_VEL
LIN {X 0,Y 516.889,Z 224.101,A -85,B 0,C 180,E1 -5064.073,E2 -5064.073} C_VEL
LIN {X 0,Y 516.909,Z 224.096,A -85,B 0,C 180,E1 -5066.659,E2 -5066.659} C_VEL
LIN {X 0,Y 516.912,Z 224.097,A -85,B 0,C 180,E1 -5069.523,E2 -5069.523} C_VEL
LIN {X 0,Y 516.896,Z 224.099,A -85,B 0,C 180,E1 -5072.543,E2 -5072.543} C_VEL
LIN {X 0,Y 516.868,Z 224.102,A -85,B 0,C 180,E1 -5075.33,E2 -5075.33} C_VEL
LIN {X 0,Y 516.883,Z 224.101,A -85,B 0,C 180,E1 -5077.943,E2 -5077.943} C_VEL
LIN {X 0,Y 516.885,Z 224.102,A -85,B 0,C 180,E1 -5080.742,E2 -5080.742} C_VEL
LIN {X 0,Y 516.885,Z 224.102,A -85,B 0,C 180,E1 -5082.831,E2 -5082.831} C_VEL
LIN {X 0,Y 516.897,Z 224.1,A -85,B 0,C 180,E1 -5085.007,E2 -5085.007} C_VEL
LIN {X 0,Y 516.915,Z 224.097,A -85,B 0,C 180,E1 -5088.399,E2 -5088.399} C_VEL
LIN {X 0,Y 516.916,Z 224.19,A -85,B 0,C 180,E1 -5091.337,E2 -5091.337} C_VEL
LIN {X 0,Y 517.987,Z 230.51,A -85,B 0,C 180,E1 -5093.828,E2 -5093.828} C_VEL
LIN {X 0,Y 518.004,Z 236.952,A -85,B 0,C 180,E1 -5096.202,E2 -5096.202} C_VEL
LIN {X 0,Y 517.631,Z 245.98,A -85,B 0,C 180,E1 -5099.393,E2 -5099.393} C_VEL
LIN {X 0,Y 517.356,Z 253.65,A -85,B 0,C 180,E1 -5102.005,E2 -5102.005} C_VEL
LIN {X 0,Y 517.148,Z 261.641,A -85,B 0,C 180,E1 -5104.654,E2 -5104.654} C_VEL
LIN {X 0,Y 516.953,Z 270.872,A -85,B 0,C 180,E1 -5107.625,E2 -5107.625} C_VEL
LIN {X 0,Y 516.764,Z 281.44,A -85,B 0,C 180,E1 -5110.95,E2 -5110.95} C_VEL
LIN {X 0,Y 516.601,Z 292.069,A -85,B 0,C 180,E1 -5114.212,E2 -5114.212} C_VEL
LIN {X 0,Y 516.532,Z 298.565,A -85,B 0,C 180,E1 -5116.112,E2 -5116.112} C_VEL
LIN {X 0,Y 518.408,Z 311.801,A -85,B 0,C 180,E1 -5116.476,E2 -5116.476} C_VEL
LIN {X 0,Y 518.131,Z 324.14,A -85,B 0,C 180,E1 -5116.918,E2 -5116.918} C_VEL
LIN {X 0,Y 517.818,Z 336.688,A -85,B 0,C 180,E1 -5117.535,E2 -5117.535} C_VEL
LIN {X 0,Y 517.488,Z 347.856,A -85,B 0,C 180,E1 -5118.246,E2 -5118.246} C_VEL
LIN {X 0,Y 517.255,Z 358.916,A -85,B 0,C 180,E1 -5119.134,E2 -5119.134} C_VEL
LIN {X 0,Y 516.957,Z 367.906,A -85,B 0,C 180,E1 -5120.018,E2 -5120.018} C_VEL
LIN {X 0,Y 516.719,Z 377.673,A -85,B 0,C 180,E1 -5121.198,E2 -5121.198} C_VEL
LIN {X 0,Y 516.547,Z 385.47,A -85,B 0,C 180,E1 -5122.377,E2 -5122.377} C_VEL
LIN {X 0,Y 516.4,Z 392.636,A -85,B 0,C 180,E1 -5123.75,E2 -5123.75} C_VEL
LIN {X 0,Y 516.313,Z 397.407,A -85,B 0,C 180,E1 -5124.924,E2 -5124.924} C_VEL
LIN {X 0,Y 516.37,Z 401.058,A -85,B 0,C 180,E1 -5126.098,E2 -5126.098} C_VEL
LIN {X 0,Y 516.282,Z 402.933,A -85,B 0,C 180,E1 -5126.879,E2 -5126.879} C_VEL
LIN {X 0,Y 516.261,Z 404.341,A -85,B 0,C 180,E1 -5127.66,E2 -5127.66} C_VEL
LIN {X 0,Y 516.165,Z 405.948,A -85,B 0,C 180,E1 -5129.22,E2 -5129.22} C_VEL
LIN {X 0,Y 516.166,Z 406.16,A -85,B 0,C 180,E1 -5130,E2 -5130} C_VEL
LIN {X 0,Y 516.192,Z 405.317,A -85,B 0,C 180,E1 -5131.561,E2 -5131.561} C_VEL
LIN {X 0,Y 516.261,Z 404.306,A -85,B 0,C 180,E1 -5132.341,E2 -5132.341} C_VEL
LIN {X 0,Y 516.282,Z 402.879,A -85,B 0,C 180,E1 -5133.121,E2 -5133.121} C_VEL
LIN {X 0,Y 516.33,Z 399.893,A -85,B 0,C 180,E1 -5134.294,E2 -5134.294} C_VEL
LIN {X 0,Y 516.397,Z 395.849,A -85,B 0,C 180,E1 -5135.467,E2 -5135.467} C_VEL
LIN {X 0,Y 516.451,Z 389.829,A -85,B 0,C 180,E1 -5136.799,E2 -5136.799} C_VEL
LIN {X 0,Y 516.586,Z 382.828,A -85,B 0,C 180,E1 -5138.016,E2 -5138.016} C_VEL
LIN {X 0,Y 516.786,Z 374.382,A -85,B 0,C 180,E1 -5139.195,E2 -5139.195} C_VEL
LIN {X 0,Y 516.994,Z 365.707,A -85,B 0,C 180,E1 -5140.179,E2 -5140.179} C_VEL
LIN {X 0,Y 517.32,Z 355.023,A -85,B 0,C 180,E1 -5141.163,E2 -5141.163} C_VEL
LIN {X 0,Y 517.522,Z 343.343,A -85,B 0,C 180,E1 -5142.028,E2 -5142.028} C_VEL
LIN {X 0,Y 517.881,Z 330.85,A -85,B 0,C 180,E1 -5142.74,E2 -5142.74} C_VEL
LIN {X 0,Y 518.187,Z 318.346,A -85,B 0,C 180,E1 -5143.281,E2 -5143.281} C_VEL
LIN {X 0,Y 518.166,Z 309.95,A -85,B 0,C 180,E1 -5143.556,E2 -5143.556} C_VEL
LIN {X 0,Y 516.636,Z 299.106,A -85,B 0,C 180,E1 -5143.854,E2 -5143.854} C_VEL
LIN {X 0,Y 516.502,Z 297.644,A -85,B 0,C 180,E1 -5143.901,E2 -5143.901} C_VEL
LIN {X 0,Y 516.588,Z 287.104,A -85,B 0,C 180,E1 -5147.008,E2 -5147.008} C_VEL
LIN {X 0,Y 516.681,Z 277.542,A -85,B 0,C 180,E1 -5149.88,E2 -5149.88} C_VEL
LIN {X 0,Y 516.846,Z 268.07,A -85,B 0,C 180,E1 -5152.801,E2 -5152.801} C_VEL
LIN {X 0,Y 517.019,Z 258.803,A -85,B 0,C 180,E1 -5155.785,E2 -5155.785} C_VEL
LIN {X 0,Y 517.177,Z 251.117,A -85,B 0,C 180,E1 -5158.4,E2 -5158.4} C_VEL
LIN {X 0,Y 517.613,Z 242.591,A -85,B 0,C 180,E1 -5161.533,E2 -5161.533} C_VEL
LIN {X 0,Y 518.075,Z 236.171,A -85,B 0,C 180,E1 -5164.157,E2 -5164.157} C_VEL
LIN {X 0,Y 518.149,Z 232.877,A -85,B 0,C 180,E1 -5165.679,E2 -5165.679} C_VEL
LIN {X 0,Y 517.821,Z 229.221,A -85,B 0,C 180,E1 -5167.644,E2 -5167.644} C_VEL
LIN {X 0,Y 517.271,Z 226.16,A -85,B 0,C 180,E1 -5169.686,E2 -5169.686} C_VEL
LIN {X 0,Y 516.917,Z 224.098,A -85,B 0,C 180,E1 -5171.601,E2 -5171.601} C_VEL
LIN {X 0,Y 516.898,Z 224.101,A -85,B 0,C 180,E1 -5175.007,E2 -5175.007} C_VEL
LIN {X 0,Y 516.917,Z 224.099,A -85,B 0,C 180,E1 -5178.399,E2 -5178.399} C_VEL
LIN {X 0,Y 516.885,Z 224.103,A -85,B 0,C 180,E1 -5181.284,E2 -5181.284} C_VEL
LIN {X 0,Y 516.874,Z 224.239,A -85,B 0,C 180,E1 -5184.22,E2 -5184.22} C_VEL
LIN {X 0,Y 516.961,Z 225.644,A -85,B 0,C 180,E1 -5186.125,E2 -5186.125} C_VEL
LIN {X 0,Y 516.831,Z 227.979,A -85,B 0,C 180,E1 -5188.948,E2 -5188.948} C_VEL
LIN {X 0,Y 516.725,Z 230.313,A -85,B 0,C 180,E1 -5191.573,E2 -5191.573} C_VEL
LIN {X 0,Y 516.678,Z 232.748,A -85,B 0,C 180,E1 -5194.197,E2 -5194.197} C_VEL
LIN {X 0,Y 516.562,Z 235.223,A -85,B 0,C 180,E1 -5196.762,E2 -5196.762} C_VEL
LIN {X 0,Y 516.476,Z 238.334,A -85,B 0,C 180,E1 -5199.873,E2 -5199.873} C_VEL
LIN {X 0,Y 516.472,Z 241.119,A -85,B 0,C 180,E1 -5202.58,E2 -5202.58} C_VEL
LIN {X 0,Y 516.408,Z 244.561,A -85,B 0,C 180,E1 -5205.82,E2 -5205.82} C_VEL
LIN {X 0,Y 516.383,Z 246.209,A -85,B 0,C 180,E1 -5207.248,E2 -5207.248} C_VEL
LIN {X 0,Y 518.324,Z 255.536,A -85,B 0,C 180,E1 -5207.547,E2 -5207.547} C_VEL
LIN {X 0,Y 518.275,Z 268.6,A -85,B 0,C 180,E1 -5208.038,E2 -5208.038} C_VEL
LIN {X 0,Y 517.994,Z 280.736,A -85,B 0,C 180,E1 -5208.654,E2 -5208.654} C_VEL
LIN {X 0,Y 517.664,Z 291.3,A -85,B 0,C 180,E1 -5209.34,E2 -5209.34} C_VEL
LIN {X 0,Y 517.393,Z 302.112,A -85,B 0,C 180,E1 -5210.224,E2 -5210.224} C_VEL
LIN {X 0,Y 517.155,Z 311.8,A -85,B 0,C 180,E1 -5211.206,E2 -5211.206} C_VEL
LIN {X 0,Y 516.862,Z 319.747,A -85,B 0,C 180,E1 -5212.185,E2 -5212.185} C_VEL
LIN {X 0,Y 516.695,Z 326.476,A -85,B 0,C 180,E1 -5213.188,E2 -5213.188} C_VEL
LIN {X 0,Y 516.573,Z 331.802,A -85,B 0,C 180,E1 -5214.144,E2 -5214.144} C_VEL
LIN {X 0,Y 516.498,Z 337.141,A -85,B 0,C 180,E1 -5215.317,E2 -5215.317} C_VEL
LIN {X 0,Y 516.434,Z 341.309,A -85,B 0,C 180,E1 -5216.489,E2 -5216.489} C_VEL
LIN {X 0,Y 516.285,Z 344.43,A -85,B 0,C 180,E1 -5217.66,E2 -5217.66} C_VEL
LIN {X 0,Y 516.205,Z 345.98,A -85,B 0,C 180,E1 -5218.44,E2 -5218.44} C_VEL
LIN {X 0,Y 516.183,Z 347.109,A -85,B 0,C 180,E1 -5219.22,E2 -5219.22} C_VEL
LIN {X 0,Y 516.175,Z 348.13,A -85,B 0,C 180,E1 -5220.78,E2 -5220.78} C_VEL
LIN {X 0,Y 516.264,Z 347.601,A -85,B 0,C 180,E1 -5222.341,E2 -5222.341} C_VEL
LIN {X 0,Y 516.356,Z 346.713,A -85,B 0,C 180,E1 -5223.121,E2 -5223.121} C_VEL
LIN {X 0,Y 516.336,Z 345.44,A -85,B 0,C 180,E1 -5223.902,E2 -5223.902} C_VEL
LIN {X 0,Y 516.297,Z 342.739,A -85,B 0,C 180,E1 -5225.076,E2 -5225.076} C_VEL
LIN {X 0,Y 516.431,Z 339.014,A -85,B 0,C 180,E1 -5226.25,E2 -5226.25} C_VEL
LIN {X 0,Y 516.504,Z 334.168,A -85,B 0,C 180,E1 -5227.427,E2 -5227.427} C_VEL
LIN {X 0,Y 516.661,Z 328.042,A -85,B 0,C 180,E1 -5228.606,E2 -5228.606} C_VEL
LIN {X 0,Y 516.84,Z 320.414,A -85,B 0,C 180,E1 -5229.787,E2 -5229.787} C_VEL
LIN {X 0,Y 517.158,Z 310.811,A -85,B 0,C 180,E1 -5230.968,E2 -5230.968} C_VEL
LIN {X 0,Y 517.363,Z 301.023,A -85,B 0,C 180,E1 -5231.944,E2 -5231.944} C_VEL
LIN {X 0,Y 517.639,Z 291.11,A -85,B 0,C 180,E1 -5232.746,E2 -5232.746} C_VEL
LIN {X 0,Y 518.034,Z 278.734,A -85,B 0,C 180,E1 -5233.534,E2 -5233.534} C_VEL
LIN {X 0,Y 518.254,Z 266.671,A -85,B 0,C 180,E1 -5234.129,E2 -5234.129} C_VEL
LIN {X 0,Y 518.281,Z 255.104,A -85,B 0,C 180,E1 -5234.552,E2 -5234.552} C_VEL
LIN {X 0,Y 516.318,Z 245.229,A -85,B 0,C 180,E1 -5234.872,E2 -5234.872} C_VEL
LIN {X 0,Y 516.326,Z 241.296,A -85,B 0,C 180,E1 -5238.244,E2 -5238.244} C_VEL
LIN {X 0,Y 516.323,Z 238.42,A -85,B 0,C 180,E1 -5240.726,E2 -5240.726} C_VEL
LIN {X 0,Y 516.342,Z 235.542,A -85,B 0,C 180,E1 -5243.249,E2 -5243.249} C_VEL
LIN {X 0,Y 516.462,Z 232.297,A -85,B 0,C 180,E1 -5246.086,E2 -5246.086} C_VEL
LIN {X 0,Y 516.419,Z 229.649,A -85,B 0,C 180,E1 -5248.445,E2 -5248.445} C_VEL
LIN {X 0,Y 516.473,Z 226.641,A -85,B 0,C 180,E1 -5251.138,E2 -5251.138} C_VEL
LIN {X 0,Y 516.471,Z 224.617,A -85,B 0,C 180,E1 -5252.978,E2 -5252.978} C_VEL
LIN {X 0,Y 516.573,Z 224.142,A -85,B 0,C 180,E1 -5253.91,E2 -5253.91} C_VEL
LIN {X 0,Y 516.807,Z 224.109,A -85,B 0,C 180,E1 -5256.752,E2 -5256.752} C_VEL
LIN {X 0,Y 516.887,Z 224.101,A -85,B 0,C 180,E1 -5259.721,E2 -5259.721} C_VEL
LIN {X 0,Y 516.912,Z 224.099,A -85,B 0,C 180,E1 -5261.776,E2 -5261.776} C_VEL
LIN {X 0,Y 516.892,Z 224.097,A -85,B 0,C 180,E1 -5264.916,E2 -5264.916} C_VEL
LIN {X 0,Y 516.266,Z 224.179,A -85,B 0,C 180,E1 -5265.566,E2 -5265.566} C_VEL
LIN {X 0,Y 513.403,Z 224.534,A -85,B 0,C 180,E1 -5266.621,E2 -5266.621} C_VEL
LIN {X 0,Y 510.959,Z 224.839,A -85,B 0,C 180,E1 -5267.471,E2 -5267.471} C_VEL
LIN {X 0,Y 509.912,Z 224.966,A -85,B 0,C 180,E1 -5268.128,E2 -5268.128} C_VEL
LIN {X 0,Y 509.83,Z 224.975,A -85,B 0,C 180,E1 -5268.35,E2 -5268.35} C_VEL
LIN {X 0,Y 509.812,Z 224.978,A -85,B 0,C 180,E1 -5271.658,E2 -5271.658} C_VEL
LIN {X 0,Y 509.81,Z 224.983,A -85,B 0,C 180,E1 -5274.62,E2 -5274.62} C_VEL
LIN {X 0,Y 509.863,Z 224.971,A -85,B 0,C 180,E1 -5277.481,E2 -5277.481} C_VEL
LIN {X 0,Y 509.862,Z 224.978,A -85,B 0,C 180,E1 -5280.274,E2 -5280.274} C_VEL
LIN {X 0,Y 509.888,Z 224.972,A -85,B 0,C 180,E1 -5283.628,E2 -5283.628} C_VEL
LIN {X 0,Y 509.827,Z 224.977,A -85,B 0,C 180,E1 -5286.436,E2 -5286.436} C_VEL
LIN {X 0,Y 509.922,Z 224.967,A -85,B 0,C 180,E1 -5289.845,E2 -5289.845} C_VEL
LIN {X 0,Y 509.873,Z 224.975,A -85,B 0,C 180,E1 -5293.174,E2 -5293.174} C_VEL
LIN {X 0,Y 509.859,Z 224.973,A -85,B 0,C 180,E1 -5295.634,E2 -5295.634} C_VEL
LIN {X 0,Y 509.915,Z 224.969,A -85,B 0,C 180,E1 -5298.874,E2 -5298.874} C_VEL
LIN {X 0,Y 509.88,Z 224.974,A -85,B 0,C 180,E1 -5302.077,E2 -5302.077} C_VEL
LIN {X 0,Y 509.933,Z 224.966,A -85,B 0,C 180,E1 -5304.464,E2 -5304.464} C_VEL
LIN {X 0,Y 510.044,Z 224.953,A -85,B 0,C 180,E1 -5307.631,E2 -5307.631} C_VEL
LIN {X 0,Y 510.042,Z 224.952,A -85,B 0,C 180,E1 -5310,E2 -5310} C_VEL
LIN {X 0,Y 510.054,Z 224.947,A -85,B 0,C 180,E1 -5312.369,E2 -5312.369} C_VEL
LIN {X 0,Y 509.733,Z 224.996,A -85,B 0,C 180,E1 -5315.538,E2 -5315.538} C_VEL
LIN {X 0,Y 509.651,Z 225.121,A -85,B 0,C 180,E1 -5315.837,E2 -5315.837} C_VEL
LIN {X 0,Y 509.606,Z 229.828,A -85,B 0,C 180,E1 -5317.927,E2 -5317.927} C_VEL
LIN {X 0,Y 509.578,Z 237.013,A -85,B 0,C 180,E1 -5321.133,E2 -5321.133} C_VEL
LIN {X 0,Y 509.519,Z 244.154,A -85,B 0,C 180,E1 -5324.376,E2 -5324.376} C_VEL
LIN {X 0,Y 509.474,Z 251.305,A -85,B 0,C 180,E1 -5327.667,E2 -5327.667} C_VEL
LIN {X 0,Y 509.356,Z 258.571,A -85,B 0,C 180,E1 -5331.023,E2 -5331.023} C_VEL
LIN {X 0,Y 509.312,Z 264.094,A -85,B 0,C 180,E1 -5333.589,E2 -5333.589} C_VEL
LIN {X 0,Y 509.352,Z 269.397,A -85,B 0,C 180,E1 -5335.982,E2 -5335.982} C_VEL
LIN {X 0,Y 510.686,Z 278.356,A -85,B 0,C 180,E1 -5336.276,E2 -5336.276} C_VEL
LIN {X 0,Y 510.495,Z 290.173,A -85,B 0,C 180,E1 -5336.777,E2 -5336.777} C_VEL
LIN {X 0,Y 510.291,Z 300.007,A -85,B 0,C 180,E1 -5337.365,E2 -5337.365} C_VEL
LIN {X 0,Y 510.129,Z 307.598,A -85,B 0,C 180,E1 -5337.932,E2 -5337.932} C_VEL
LIN {X 0,Y 509.975,Z 315.389,A -85,B 0,C 180,E1 -5338.644,E2 -5338.644} C_VEL
LIN {X 0,Y 509.772,Z 323.032,A -85,B 0,C 180,E1 -5339.501,E2 -5339.501} C_VEL
LIN {X 0,Y 509.585,Z 329.851,A -85,B 0,C 180,E1 -5340.454,E2 -5340.454} C_VEL
LIN {X 0,Y 509.433,Z 336.342,A -85,B 0,C 180,E1 -5341.617,E2 -5341.617} C_VEL
LIN {X 0,Y 509.281,Z 340.841,A -85,B 0,C 180,E1 -5342.67,E2 -5342.67} C_VEL
LIN {X 0,Y 509.266,Z 343.619,A -85,B 0,C 180,E1 -5343.505,E2 -5343.505} C_VEL
LIN {X 0,Y 509.203,Z 346.015,A -85,B 0,C 180,E1 -5344.463,E2 -5344.463} C_VEL
LIN {X 0,Y 509.136,Z 347.686,A -85,B 0,C 180,E1 -5345.469,E2 -5345.469} C_VEL
LIN {X 0,Y 509.101,Z 348.673,A -85,B 0,C 180,E1 -5346.805,E2 -5346.805} C_VEL
LIN {X 0,Y 509.092,Z 348.307,A -85,B 0,C 180,E1 -5348.104,E2 -5348.104} C_VEL
LIN {X 0,Y 509.173,Z 346.47,A -85,B 0,C 180,E1 -5349.415,E2 -5349.415} C_VEL
LIN {X 0,Y 509.25,Z 343.568,A -85,B 0,C 180,E1 -5350.62,E2 -5350.62} C_VEL
LIN {X 0,Y 509.363,Z 339.295,A -85,B 0,C 180,E1 -5351.834,E2 -5351.834} C_VEL
LIN {X 0,Y 509.47,Z 333.582,A -85,B 0,C 180,E1 -5353.019,E2 -5353.019} C_VEL
LIN {X 0,Y 509.62,Z 327.215,A -85,B 0,C 180,E1 -5354.04,E2 -5354.04} C_VEL
LIN {X 0,Y 509.869,Z 319.673,A -85,B 0,C 180,E1 -5355.007,E2 -5355.007} C_VEL
LIN {X 0,Y 510.081,Z 310.236,A -85,B 0,C 180,E1 -5355.945,E2 -5355.945} C_VEL
LIN {X 0,Y 510.291,Z 301.699,A -85,B 0,C 180,E1 -5356.615,E2 -5356.615} C_VEL
LIN {X 0,Y 510.462,Z 293.197,A -85,B 0,C 180,E1 -5357.15,E2 -5357.15} C_VEL
LIN {X 0,Y 510.649,Z 283.426,A -85,B 0,C 180,E1 -5357.627,E2 -5357.627} C_VEL
LIN {X 0,Y 510.466,Z 276.234,A -85,B 0,C 180,E1 -5357.895,E2 -5357.895} C_VEL
LIN {X 0,Y 509.316,Z 269.408,A -85,B 0,C 180,E1 -5358.124,E2 -5358.124} C_VEL
LIN {X 0,Y 509.37,Z 262.948,A -85,B 0,C 180,E1 -5361.113,E2 -5361.113} C_VEL
LIN {X 0,Y 509.353,Z 257.538,A -85,B 0,C 180,E1 -5363.607,E2 -5363.607} C_VEL
LIN {X 0,Y 509.49,Z 251.06,A -85,B 0,C 180,E1 -5366.511,E2 -5366.511} C_VEL
LIN {X 0,Y 509.464,Z 244.98,A -85,B 0,C 180,E1 -5369.309,E2 -5369.309} C_VEL
LIN {X 0,Y 509.506,Z 238.815,A -85,B 0,C 180,E1 -5372.031,E2 -5372.031} C_VEL
LIN {X 0,Y 509.529,Z 231.619,A -85,B 0,C 180,E1 -5375.122,E2 -5375.122} C_VEL
LIN {X 0,Y 509.63,Z 225.01,A -85,B 0,C 180,E1 -5377.965,E2 -5377.965} C_VEL
LIN {X 0,Y 509.891,Z 224.975,A -85,B 0,C 180,E1 -5379.843,E2 -5379.843} C_VEL
LIN {X 0,Y 509.875,Z 224.975,A -85,B 0,C 180,E1 -5383.174,E2 -5383.174} C_VEL
LIN {X 0,Y 509.865,Z 224.976,A -85,B 0,C 180,E1 -5385.634,E2 -5385.634} C_VEL
LIN {X 0,Y 509.917,Z 224.969,A -85,B 0,C 180,E1 -5388.874,E2 -5388.874} C_VEL
LIN {X 0,Y 509.955,Z 224.965,A -85,B 0,C 180,E1 -5392.078,E2 -5392.078} C_VEL
LIN {X 0,Y 509.971,Z 224.963,A -85,B 0,C 180,E1 -5394.464,E2 -5394.464} C_VEL
LIN {X 0,Y 510.058,Z 224.953,A -85,B 0,C 180,E1 -5397.631,E2 -5397.631} C_VEL
LIN {X 0,Y 510.066,Z 224.95,A -85,B 0,C 180,E1 -5400.789,E2 -5400.789} C_VEL
LIN {X 0,Y 509.955,Z 224.964,A -85,B 0,C 180,E1 -5403.16,E2 -5403.16} C_VEL
LIN {X 0,Y 509.939,Z 224.967,A -85,B 0,C 180,E1 -5406.33,E2 -5406.33} C_VEL
LIN {X 0,Y 509.915,Z 224.969,A -85,B 0,C 180,E1 -5408.72,E2 -5408.72} C_VEL
LIN {X 0,Y 509.908,Z 224.972,A -85,B 0,C 180,E1 -5411.932,E2 -5411.932} C_VEL
LIN {X 0,Y 509.897,Z 224.972,A -85,B 0,C 180,E1 -5415.242,E2 -5415.242} C_VEL
LIN {X 0,Y 509.864,Z 224.974,A -85,B 0,C 180,E1 -5418.484,E2 -5418.484} C_VEL
LIN {X 0,Y 509.853,Z 224.976,A -85,B 0,C 180,E1 -5421.002,E2 -5421.002} C_VEL
LIN {X 0,Y 509.823,Z 224.981,A -85,B 0,C 180,E1 -5423.564,E2 -5423.564} C_VEL
LIN {X 0,Y 509.888,Z 224.973,A -85,B 0,C 180,E1 -5426.372,E2 -5426.372} C_VEL
LIN {X 0,Y 509.877,Z 224.974,A -85,B 0,C 180,E1 -5428.844,E2 -5428.844} C_VEL
LIN {X 0,Y 509.821,Z 224.98,A -85,B 0,C 180,E1 -5431.59,E2 -5431.59} C_VEL
LIN {X 0,Y 509.84,Z 224.979,A -85,B 0,C 180,E1 -5434.414,E2 -5434.414} C_VEL
LIN {X 0,Y 509.819,Z 224.98,A -85,B 0,C 180,E1 -5437.341,E2 -5437.341} C_VEL
LIN {X 0,Y 509.84,Z 224.979,A -85,B 0,C 180,E1 -5440.382,E2 -5440.382} C_VEL
LIN {X 0,Y 509.825,Z 224.982,A -85,B 0,C 180,E1 -5443.062,E2 -5443.062} C_VEL
LIN {X 0,Y 509.824,Z 224.981,A -85,B 0,C 180,E1 -5445.793,E2 -5445.793} C_VEL
LIN {X 0,Y 509.857,Z 224.977,A -85,B 0,C 180,E1 -5448.574,E2 -5448.574} C_VEL
LIN {X 0,Y 509.861,Z 225.083,A -85,B 0,C 180,E1 -5451.094,E2 -5451.094} C_VEL
LIN {X 0,Y 511.005,Z 231.68,A -85,B 0,C 180,E1 -5453.744,E2 -5453.744} C_VEL
LIN {X 0,Y 511.037,Z 238.124,A -85,B 0,C 180,E1 -5456.153,E2 -5456.153} C_VEL
LIN {X 0,Y 510.634,Z 247.152,A -85,B 0,C 180,E1 -5459.387,E2 -5459.387} C_VEL
LIN {X 0,Y 510.25,Z 256.247,A -85,B 0,C 180,E1 -5462.521,E2 -5462.521} C_VEL
LIN {X 0,Y 510.081,Z 264.899,A -85,B 0,C 180,E1 -5465.418,E2 -5465.418} C_VEL
LIN {X 0,Y 509.823,Z 274.603,A -85,B 0,C 180,E1 -5468.574,E2 -5468.574} C_VEL
LIN {X 0,Y 509.667,Z 283.852,A -85,B 0,C 180,E1 -5471.509,E2 -5471.509} C_VEL
LIN {X 0,Y 509.483,Z 294.853,A -85,B 0,C 180,E1 -5474.93,E2 -5474.93} C_VEL
LIN {X 0,Y 509.443,Z 297.991,A -85,B 0,C 180,E1 -5475.902,E2 -5475.902} C_VEL
LIN {X 0,Y 511.442,Z 312.863,A -85,B 0,C 180,E1 -5476.339,E2 -5476.339} C_VEL
LIN {X 0,Y 511.136,Z 325.864,A -85,B 0,C 180,E1 -5476.837,E2 -5476.837} C_VEL
LIN {X 0,Y 510.799,Z 337.891,A -85,B 0,C 180,E1 -5477.461,E2 -5477.461} C_VEL
LIN {X 0,Y 510.448,Z 348.728,A -85,B 0,C 180,E1 -5478.182,E2 -5478.182} C_VEL
LIN {X 0,Y 510.212,Z 359.521,A -85,B 0,C 180,E1 -5479.082,E2 -5479.082} C_VEL
LIN {X 0,Y 509.871,Z 369.24,A -85,B 0,C 180,E1 -5480.079,E2 -5480.079} C_VEL
LIN {X 0,Y 509.676,Z 377.227,A -85,B 0,C 180,E1 -5481.076,E2 -5481.076} C_VEL
LIN {X 0,Y 509.473,Z 385.043,A -85,B 0,C 180,E1 -5482.27,E2 -5482.27} C_VEL
LIN {X 0,Y 509.308,Z 392.22,A -85,B 0,C 180,E1 -5483.662,E2 -5483.662} C_VEL
LIN {X 0,Y 509.246,Z 397.003,A -85,B 0,C 180,E1 -5484.853,E2 -5484.853} C_VEL
LIN {X 0,Y 509.275,Z 400.659,A -85,B 0,C 180,E1 -5486.044,E2 -5486.044} C_VEL
LIN {X 0,Y 509.201,Z 402.538,A -85,B 0,C 180,E1 -5486.835,E2 -5486.835} C_VEL
LIN {X 0,Y 509.19,Z 403.949,A -85,B 0,C 180,E1 -5487.627,E2 -5487.627} C_VEL
LIN {X 0,Y 509.078,Z 405.554,A -85,B 0,C 180,E1 -5489.209,E2 -5489.209} C_VEL
LIN {X 0,Y 509.078,Z 405.763,A -85,B 0,C 180,E1 -5490,E2 -5490} C_VEL
LIN {X 0,Y 509.112,Z 404.913,A -85,B 0,C 180,E1 -5491.582,E2 -5491.582} C_VEL
LIN {X 0,Y 509.19,Z 403.893,A -85,B 0,C 180,E1 -5492.373,E2 -5492.373} C_VEL
LIN {X 0,Y 509.201,Z 402.457,A -85,B 0,C 180,E1 -5493.165,E2 -5493.165} C_VEL
LIN {X 0,Y 509.221,Z 399.453,A -85,B 0,C 180,E1 -5494.354,E2 -5494.354} C_VEL
LIN {X 0,Y 509.309,Z 395.391,A -85,B 0,C 180,E1 -5495.543,E2 -5495.543} C_VEL
LIN {X 0,Y 509.373,Z 389.598,A -85,B 0,C 180,E1 -5496.845,E2 -5496.845} C_VEL
LIN {X 0,Y 509.503,Z 382.309,A -85,B 0,C 180,E1 -5498.128,E2 -5498.128} C_VEL
LIN {X 0,Y 509.735,Z 373.833,A -85,B 0,C 180,E1 -5499.323,E2 -5499.323} C_VEL
LIN {X 0,Y 509.967,Z 365.119,A -85,B 0,C 180,E1 -5500.321,E2 -5500.321} C_VEL
LIN {X 0,Y 510.3,Z 354.397,A -85,B 0,C 180,E1 -5501.318,E2 -5501.318} C_VEL
LIN {X 0,Y 510.502,Z 343.681,A -85,B 0,C 180,E1 -5502.127,E2 -5502.127} C_VEL
LIN {X 0,Y 510.862,Z 332.132,A -85,B 0,C 180,E1 -5502.817,E2 -5502.817} C_VEL
LIN {X 0,Y 511.21,Z 318.887,A -85,B 0,C 180,E1 -5503.415,E2 -5503.415} C_VEL
LIN {X 0,Y 511.192,Z 310.753,A -85,B 0,C 180,E1 -5503.7,E2 -5503.7} C_VEL
LIN {X 0,Y 509.695,Z 299.563,A -85,B 0,C 180,E1 -5504.024,E2 -5504.024} C_VEL
LIN {X 0,Y 509.406,Z 297.141,A -85,B 0,C 180,E1 -5504.099,E2 -5504.099} C_VEL
LIN {X 0,Y 509.531,Z 286.647,A -85,B 0,C 180,E1 -5507.251,E2 -5507.251} C_VEL
LIN {X 0,Y 509.668,Z 275.68,A -85,B 0,C 180,E1 -5510.623,E2 -5510.623} C_VEL
LIN {X 0,Y 509.78,Z 267.74,A -85,B 0,C 180,E1 -5513.136,E2 -5513.136} C_VEL
LIN {X 0,Y 510.031,Z 257.864,A -85,B 0,C 180,E1 -5516.405,E2 -5516.405} C_VEL
LIN {X 0,Y 510.246,Z 249.778,A -85,B 0,C 180,E1 -5519.273,E2 -5519.273} C_VEL
LIN {X 0,Y 510.677,Z 242.686,A -85,B 0,C 180,E1 -5521.995,E2 -5521.995} C_VEL
LIN {X 0,Y 511.149,Z 236.997,A -85,B 0,C 180,E1 -5524.415,E2 -5524.415} C_VEL
LIN {X 0,Y 511.129,Z 233.243,A -85,B 0,C 180,E1 -5526.246,E2 -5526.246} C_VEL
LIN {X 0,Y 510.717,Z 229.659,A -85,B 0,C 180,E1 -5528.336,E2 -5528.336} C_VEL
LIN {X 0,Y 510.123,Z 226.492,A -85,B 0,C 180,E1 -5530.735,E2 -5530.735} C_VEL
LIN {X 0,Y 509.836,Z 224.98,A -85,B 0,C 180,E1 -5532.49,E2 -5532.49} C_VEL
LIN {X 0,Y 509.842,Z 224.98,A -85,B 0,C 180,E1 -5535.33,E2 -5535.33} C_VEL
LIN {X 0,Y 509.859,Z 224.978,A -85,B 0,C 180,E1 -5538.575,E2 -5538.575} C_VEL
LIN {X 0,Y 509.855,Z 224.979,A -85,B 0,C 180,E1 -5541.787,E2 -5541.787} C_VEL
LIN {X 0,Y 509.828,Z 225.079,A -85,B 0,C 180,E1 -5543.647,E2 -5543.647} C_VEL
LIN {X 0,Y 509.927,Z 226.514,A -85,B 0,C 180,E1 -5545.787,E2 -5545.787} C_VEL
LIN {X 0,Y 509.811,Z 228.558,A -85,B 0,C 180,E1 -5548.409,E2 -5548.409} C_VEL
LIN {X 0,Y 509.725,Z 230.883,A -85,B 0,C 180,E1 -5551.146,E2 -5551.146} C_VEL
LIN {X 0,Y 509.636,Z 233.281,A -85,B 0,C 180,E1 -5553.814,E2 -5553.814} C_VEL
LIN {X 0,Y 509.544,Z 235.745,A -85,B 0,C 180,E1 -5556.422,E2 -5556.422} C_VEL
LIN {X 0,Y 509.428,Z 238.233,A -85,B 0,C 180,E1 -5558.98,E2 -5558.98} C_VEL
LIN {X 0,Y 509.419,Z 241.618,A -85,B 0,C 180,E1 -5562.331,E2 -5562.331} C_VEL
LIN {X 0,Y 509.368,Z 245.058,A -85,B 0,C 180,E1 -5565.62,E2 -5565.62} C_VEL
LIN {X 0,Y 509.321,Z 246.608,A -85,B 0,C 180,E1 -5567.055,E2 -5567.055} C_VEL
LIN {X 0,Y 511.517,Z 257.02,A -85,B 0,C 180,E1 -5567.406,E2 -5567.406} C_VEL
LIN {X 0,Y 511.324,Z 270.319,A -85,B 0,C 180,E1 -5567.928,E2 -5567.928} C_VEL
LIN {X 0,Y 511.055,Z 282.897,A -85,B 0,C 180,E1 -5568.598,E2 -5568.598} C_VEL
LIN {X 0,Y 510.655,Z 294.349,A -85,B 0,C 180,E1 -5569.393,E2 -5569.393} C_VEL
LIN {X 0,Y 510.347,Z 304.676,A -85,B 0,C 180,E1 -5570.288,E2 -5570.288} C_VEL
LIN {X 0,Y 510.096,Z 313.991,A -85,B 0,C 180,E1 -5571.283,E2 -5571.283} C_VEL
LIN {X 0,Y 509.777,Z 322.966,A -85,B 0,C 180,E1 -5572.474,E2 -5572.474} C_VEL
LIN {X 0,Y 509.627,Z 330.188,A -85,B 0,C 180,E1 -5573.666,E2 -5573.666} C_VEL
LIN {X 0,Y 509.441,Z 335.969,A -85,B 0,C 180,E1 -5574.855,E2 -5574.855} C_VEL
LIN {X 0,Y 509.335,Z 340.511,A -85,B 0,C 180,E1 -5576.044,E2 -5576.044} C_VEL
LIN {X 0,Y 509.355,Z 342.903,A -85,B 0,C 180,E1 -5576.836,E2 -5576.836} C_VEL
LIN {X 0,Y 509.216,Z 344.863,A -85,B 0,C 180,E1 -5577.627,E2 -5577.627} C_VEL
LIN {X 0,Y 509.126,Z 346.408,A -85,B 0,C 180,E1 -5578.418,E2 -5578.418} C_VEL
LIN {X 0,Y 509.096,Z 347.528,A -85,B 0,C 180,E1 -5579.209,E2 -5579.209} C_VEL
LIN {X 0,Y 509.088,Z 348.532,A -85,B 0,C 180,E1 -5580.791,E2 -5580.791} C_VEL
LIN {X 0,Y 509.114,Z 348.457,A -85,B 0,C 180,E1 -5581.582,E2 -5581.582} C_VEL
LIN {X 0,Y 509.195,Z 347.978,A -85,B 0,C 180,E1 -5582.373,E2 -5582.373} C_VEL
LIN {X 0,Y 509.279,Z 347.079,A -85,B 0,C 180,E1 -5583.164,E2 -5583.164} C_VEL
LIN {X 0,Y 509.263,Z 345.789,A -85,B 0,C 180,E1 -5583.957,E2 -5583.957} C_VEL
LIN {X 0,Y 509.232,Z 343.064,A -85,B 0,C 180,E1 -5585.147,E2 -5585.147} C_VEL
LIN {X 0,Y 509.336,Z 339.311,A -85,B 0,C 180,E1 -5586.338,E2 -5586.338} C_VEL
LIN {X 0,Y 509.454,Z 334.429,A -85,B 0,C 180,E1 -5587.531,E2 -5587.531} C_VEL
LIN {X 0,Y 509.627,Z 328.268,A -85,B 0,C 180,E1 -5588.725,E2 -5588.725} C_VEL
LIN {X 0,Y 509.805,Z 320.591,A -85,B 0,C 180,E1 -5589.923,E2 -5589.923} C_VEL
LIN {X 0,Y 510.162,Z 310.935,A -85,B 0,C 180,E1 -5591.12,E2 -5591.12} C_VEL
LIN {X 0,Y 510.367,Z 301.812,A -85,B 0,C 180,E1 -5592.043,E2 -5592.043} C_VEL
LIN {X 0,Y 510.698,Z 291.101,A -85,B 0,C 180,E1 -5592.922,E2 -5592.922} C_VEL
LIN {X 0,Y 511.131,Z 278.654,A -85,B 0,C 180,E1 -5593.721,E2 -5593.721} C_VEL
LIN {X 0,Y 511.345,Z 266.486,A -85,B 0,C 180,E1 -5594.324,E2 -5594.324} C_VEL
LIN {X 0,Y 511.391,Z 256.18,A -85,B 0,C 180,E1 -5594.707,E2 -5594.707} C_VEL
LIN {X 0,Y 509.234,Z 245.559,A -85,B 0,C 180,E1 -5595.056,E2 -5595.056} C_VEL
LIN {X 0,Y 509.283,Z 242.39,A -85,B 0,C 180,E1 -5597.788,E2 -5597.788} C_VEL
LIN {X 0,Y 509.274,Z 239.576,A -85,B 0,C 180,E1 -5600.214,E2 -5600.214} C_VEL
LIN {X 0,Y 509.241,Z 236.694,A -85,B 0,C 180,E1 -5602.733,E2 -5602.733} C_VEL
LIN {X 0,Y 509.351,Z 233.755,A -85,B 0,C 180,E1 -5605.324,E2 -5605.324} C_VEL
LIN {X 0,Y 509.366,Z 230.771,A -85,B 0,C 180,E1 -5607.987,E2 -5607.987} C_VEL
LIN {X 0,Y 509.399,Z 227.225,A -85,B 0,C 180,E1 -5611.196,E2 -5611.196} C_VEL
LIN {X 0,Y 509.403,Z 225.569,A -85,B 0,C 180,E1 -5612.691,E2 -5612.691} C_VEL
LIN {X 0,Y 509.474,Z 225.026,A -85,B 0,C 180,E1 -5613.49,E2 -5613.49} C_VEL
LIN {X 0,Y 509.748,Z 224.99,A -85,B 0,C 180,E1 -5616.36,E2 -5616.36} C_VEL
LIN {X 0,Y 509.851,Z 224.975,A -85,B 0,C 180,E1 -5619.352,E2 -5619.352} C_VEL
LIN {X 0,Y 509.821,Z 224.978,A -85,B 0,C 180,E1 -5622.492,E2 -5622.492} C_VEL
LIN {X 0,Y 509.843,Z 224.98,A -85,B 0,C 180,E1 -5625.33,E2 -5625.33} C_VEL
LIN {X 0,Y 509.83,Z 224.975,A -85,B 0,C 180,E1 -5628.35,E2 -5628.35} C_VEL
LIN {X 0,Y 509.168,Z 225.063,A -85,B 0,C 180,E1 -5629.01,E2 -5629.01} C_VEL
LIN {X 0,Y 506.299,Z 225.417,A -85,B 0,C 180,E1 -5630.079,E2 -5630.079} C_VEL
LIN {X 0,Y 503.872,Z 225.724,A -85,B 0,C 180,E1 -5630.941,E2 -5630.941} C_VEL
LIN {X 0,Y 502.835,Z 225.847,A -85,B 0,C 180,E1 -5631.607,E2 -5631.607} C_VEL
LIN {X 0,Y 502.753,Z 225.856,A -85,B 0,C 180,E1 -5631.833,E2 -5631.833} C_VEL
LIN {X 0,Y 502.785,Z 225.856,A -85,B 0,C 180,E1 -5635.033,E2 -5635.033} C_VEL
LIN {X 0,Y 502.786,Z 225.854,A -85,B 0,C 180,E1 -5637.915,E2 -5637.915} C_VEL
LIN {X 0,Y 502.817,Z 225.851,A -85,B 0,C 180,E1 -5640.711,E2 -5640.711} C_VEL
LIN {X 0,Y 502.849,Z 225.847,A -85,B 0,C 180,E1 -5643.443,E2 -5643.443} C_VEL
LIN {X 0,Y 502.779,Z 225.858,A -85,B 0,C 180,E1 -5646.085,E2 -5646.085} C_VEL
LIN {X 0,Y 502.788,Z 225.854,A -85,B 0,C 180,E1 -5648.689,E2 -5648.689} C_VEL
LIN {X 0,Y 502.83,Z 225.852,A -85,B 0,C 180,E1 -5651.248,E2 -5651.248} C_VEL
LIN {X 0,Y 502.853,Z 225.848,A -85,B 0,C 180,E1 -5654.6,E2 -5654.6} C_VEL
LIN {X 0,Y 502.881,Z 225.843,A -85,B 0,C 180,E1 -5658.039,E2 -5658.039} C_VEL
LIN {X 0,Y 502.852,Z 225.846,A -85,B 0,C 180,E1 -5661.156,E2 -5661.156} C_VEL
LIN {X 0,Y 502.852,Z 225.846,A -85,B 0,C 180,E1 -5663.58,E2 -5663.58} C_VEL
LIN {X 0,Y 502.743,Z 225.865,A -85,B 0,C 180,E1 -5665.992,E2 -5665.992} C_VEL
LIN {X 0,Y 503.011,Z 225.828,A -85,B 0,C 180,E1 -5667.598,E2 -5667.598} C_VEL
LIN {X 0,Y 503.011,Z 225.828,A -85,B 0,C 180,E1 -5670,E2 -5670} C_VEL
LIN {X 0,Y 503.023,Z 225.823,A -85,B 0,C 180,E1 -5672.402,E2 -5672.402} C_VEL
LIN {X 0,Y 502.674,Z 225.876,A -85,B 0,C 180,E1 -5675.616,E2 -5675.616} C_VEL
LIN {X 0,Y 502.594,Z 225.911,A -85,B 0,C 180,E1 -5675.819,E2 -5675.819} C_VEL
LIN {X 0,Y 502.542,Z 230.881,A -85,B 0,C 180,E1 -5678.039,E2 -5678.039} C_VEL
LIN {X 0,Y 502.524,Z 238.103,A -85,B 0,C 180,E1 -5681.291,E2 -5681.291} C_VEL
LIN {X 0,Y 502.473,Z 245.33,A -85,B 0,C 180,E1 -5684.582,E2 -5684.582} C_VEL
LIN {X 0,Y 502.405,Z 252.678,A -85,B 0,C 180,E1 -5687.966,E2 -5687.966} C_VEL
LIN {X 0,Y 502.318,Z 258.07,A -85,B 0,C 180,E1 -5690.474,E2 -5690.474} C_VEL
LIN {X 0,Y 502.239,Z 263.653,A -85,B 0,C 180,E1 -5693.067,E2 -5693.067} C_VEL
LIN {X 0,Y 502.29,Z 269.545,A -85,B 0,C 180,E1 -5695.813,E2 -5695.813} C_VEL
LIN {X 0,Y 503.708,Z 279.795,A -85,B 0,C 180,E1 -5696.166,E2 -5696.166} C_VEL
LIN {X 0,Y 503.516,Z 291.801,A -85,B 0,C 180,E1 -5696.708,E2 -5696.708} C_VEL
LIN {X 0,Y 503.304,Z 300.185,A -85,B 0,C 180,E1 -5697.219,E2 -5697.219} C_VEL
LIN {X 0,Y 503.105,Z 309.082,A -85,B 0,C 180,E1 -5697.903,E2 -5697.903} C_VEL
LIN {X 0,Y 502.936,Z 316.392,A -85,B 0,C 180,E1 -5698.595,E2 -5698.595} C_VEL
LIN {X 0,Y 502.742,Z 324.146,A -85,B 0,C 180,E1 -5699.49,E2 -5699.49} C_VEL
LIN {X 0,Y 502.526,Z 330.862,A -85,B 0,C 180,E1 -5700.462,E2 -5700.462} C_VEL
LIN {X 0,Y 502.382,Z 336.148,A -85,B 0,C 180,E1 -5701.421,E2 -5701.421} C_VEL
LIN {X 0,Y 502.214,Z 340.848,A -85,B 0,C 180,E1 -5702.511,E2 -5702.511} C_VEL
LIN {X 0,Y 502.2,Z 344.272,A -85,B 0,C 180,E1 -5703.558,E2 -5703.558} C_VEL
LIN {X 0,Y 502.145,Z 346.202,A -85,B 0,C 180,E1 -5704.334,E2 -5704.334} C_VEL
LIN {X 0,Y 502.071,Z 347.534,A -85,B 0,C 180,E1 -5705.024,E2 -5705.024} C_VEL
LIN {X 0,Y 502.026,Z 348.71,A -85,B 0,C 180,E1 -5706.013,E2 -5706.013} C_VEL
LIN {X 0,Y 502.012,Z 349.128,A -85,B 0,C 180,E1 -5707.062,E2 -5707.062} C_VEL
LIN {X 0,Y 502.025,Z 348.401,A -85,B 0,C 180,E1 -5708.375,E2 -5708.375} C_VEL
LIN {X 0,Y 502.057,Z 347.596,A -85,B 0,C 180,E1 -5709.045,E2 -5709.045} C_VEL
LIN {X 0,Y 502.15,Z 345.568,A -85,B 0,C 180,E1 -5710.076,E2 -5710.076} C_VEL
LIN {X 0,Y 502.218,Z 342.567,A -85,B 0,C 180,E1 -5711.126,E2 -5711.126} C_VEL
LIN {X 0,Y 502.296,Z 338.433,A -85,B 0,C 180,E1 -5712.191,E2 -5712.191} C_VEL
LIN {X 0,Y 502.433,Z 333.022,A -85,B 0,C 180,E1 -5713.268,E2 -5713.268} C_VEL
LIN {X 0,Y 502.643,Z 326.103,A -85,B 0,C 180,E1 -5714.355,E2 -5714.355} C_VEL
LIN {X 0,Y 502.903,Z 318.164,A -85,B 0,C 180,E1 -5715.327,E2 -5715.327} C_VEL
LIN {X 0,Y 503.089,Z 310.342,A -85,B 0,C 180,E1 -5716.091,E2 -5716.091} C_VEL
LIN {X 0,Y 503.314,Z 301.925,A -85,B 0,C 180,E1 -5716.758,E2 -5716.758} C_VEL
LIN {X 0,Y 503.494,Z 293.364,A -85,B 0,C 180,E1 -5717.301,E2 -5717.301} C_VEL
LIN {X 0,Y 503.699,Z 282.531,A -85,B 0,C 180,E1 -5717.829,E2 -5717.829} C_VEL
LIN {X 0,Y 503.419,Z 276.233,A -85,B 0,C 180,E1 -5718.059,E2 -5718.059} C_VEL
LIN {X 0,Y 502.268,Z 269.769,A -85,B 0,C 180,E1 -5718.277,E2 -5718.277} C_VEL
LIN {X 0,Y 502.331,Z 262.635,A -85,B 0,C 180,E1 -5721.581,E2 -5721.581} C_VEL
LIN {X 0,Y 502.345,Z 255.193,A -85,B 0,C 180,E1 -5724.998,E2 -5724.998} C_VEL
LIN {X 0,Y 502.412,Z 250.676,A -85,B 0,C 180,E1 -5727.068,E2 -5727.068} C_VEL
LIN {X 0,Y 502.436,Z 244.773,A -85,B 0,C 180,E1 -5729.764,E2 -5729.764} C_VEL
LIN {X 0,Y 502.441,Z 238.474,A -85,B 0,C 180,E1 -5732.51,E2 -5732.51} C_VEL
LIN {X 0,Y 502.492,Z 231.828,A -85,B 0,C 180,E1 -5735.383,E2 -5735.383} C_VEL
LIN {X 0,Y 502.563,Z 225.891,A -85,B 0,C 180,E1 -5737.924,E2 -5737.924} C_VEL
LIN {X 0,Y 502.811,Z 225.855,A -85,B 0,C 180,E1 -5740.399,E2 -5740.399} C_VEL
LIN {X 0,Y 502.821,Z 225.853,A -85,B 0,C 180,E1 -5742.931,E2 -5742.931} C_VEL
LIN {X 0,Y 502.847,Z 225.849,A -85,B 0,C 180,E1 -5745.429,E2 -5745.429} C_VEL
LIN {X 0,Y 502.881,Z 225.846,A -85,B 0,C 180,E1 -5748.717,E2 -5748.717} C_VEL
LIN {X 0,Y 502.905,Z 225.844,A -85,B 0,C 180,E1 -5751.967,E2 -5751.967} C_VEL
LIN {X 0,Y 502.872,Z 225.848,A -85,B 0,C 180,E1 -5755.19,E2 -5755.19} C_VEL
LIN {X 0,Y 503.028,Z 225.829,A -85,B 0,C 180,E1 -5757.598,E2 -5757.598} C_VEL
LIN {X 0,Y 503.031,Z 225.828,A -85,B 0,C 180,E1 -5760,E2 -5760} C_VEL
LIN {X 0,Y 503.028,Z 225.829,A -85,B 0,C 180,E1 -5762.402,E2 -5762.402} C_VEL
LIN {X 0,Y 502.929,Z 225.839,A -85,B 0,C 180,E1 -5765.614,E2 -5765.614} C_VEL
LIN {X 0,Y 502.873,Z 225.846,A -85,B 0,C 180,E1 -5768.843,E2 -5768.843} C_VEL
LIN {X 0,Y 502.849,Z 225.851,A -85,B 0,C 180,E1 -5772.102,E2 -5772.102} C_VEL
LIN {X 0,Y 502.852,Z 225.85,A -85,B 0,C 180,E1 -5775.4,E2 -5775.4} C_VEL
LIN {X 0,Y 502.829,Z 225.851,A -85,B 0,C 180,E1 -5778.752,E2 -5778.752} C_VEL
LIN {X 0,Y 502.786,Z 225.858,A -85,B 0,C 180,E1 -5781.311,E2 -5781.311} C_VEL
LIN {X 0,Y 502.773,Z 225.86,A -85,B 0,C 180,E1 -5783.915,E2 -5783.915} C_VEL
LIN {X 0,Y 502.839,Z 225.849,A -85,B 0,C 180,E1 -5786.568,E2 -5786.568} C_VEL
LIN {X 0,Y 502.825,Z 225.851,A -85,B 0,C 180,E1 -5789.288,E2 -5789.288} C_VEL
LIN {X 0,Y 502.784,Z 225.858,A -85,B 0,C 180,E1 -5792.085,E2 -5792.085} C_VEL
LIN {X 0,Y 502.798,Z 225.855,A -85,B 0,C 180,E1 -5794.966,E2 -5794.966} C_VEL
LIN {X 0,Y 502.795,Z 225.856,A -85,B 0,C 180,E1 -5797.954,E2 -5797.954} C_VEL
LIN {X 0,Y 502.822,Z 225.852,A -85,B 0,C 180,E1 -5801.066,E2 -5801.066} C_VEL
LIN {X 0,Y 502.788,Z 225.857,A -85,B 0,C 180,E1 -5804.53,E2 -5804.53} C_VEL
LIN {X 0,Y 502.797,Z 225.857,A -85,B 0,C 180,E1 -5807.861,E2 -5807.861} C_VEL
LIN {X 0,Y 502.809,Z 225.907,A -85,B 0,C 180,E1 -5810.831,E2 -5810.831} C_VEL
LIN {X 0,Y 503.99,Z 232.705,A -85,B 0,C 180,E1 -5813.602,E2 -5813.602} C_VEL
LIN {X 0,Y 504.081,Z 238.248,A -85,B 0,C 180,E1 -5815.721,E2 -5815.721} C_VEL
LIN {X 0,Y 503.697,Z 247.025,A -85,B 0,C 180,E1 -5818.919,E2 -5818.919} C_VEL
LIN {X 0,Y 503.289,Z 256.086,A -85,B 0,C 180,E1 -5822.108,E2 -5822.108} C_VEL
LIN {X 0,Y 503.059,Z 265.2,A -85,B 0,C 180,E1 -5825.221,E2 -5825.221} C_VEL
LIN {X 0,Y 502.779,Z 274.385,A -85,B 0,C 180,E1 -5828.258,E2 -5828.258} C_VEL
LIN {X 0,Y 502.62,Z 283.59,A -85,B 0,C 180,E1 -5831.24,E2 -5831.24} C_VEL
LIN {X 0,Y 502.429,Z 294.162,A -85,B 0,C 180,E1 -5834.587,E2 -5834.587} C_VEL
LIN {X 0,Y 502.343,Z 297.675,A -85,B 0,C 180,E1 -5835.699,E2 -5835.699} C_VEL
LIN {X 0,Y 504.5,Z 313.094,A -85,B 0,C 180,E1 -5836.173,E2 -5836.173} C_VEL
LIN {X 0,Y 504.173,Z 326.43,A -85,B 0,C 180,E1 -5836.703,E2 -5836.703} C_VEL
LIN {X 0,Y 503.795,Z 338.913,A -85,B 0,C 180,E1 -5837.379,E2 -5837.379} C_VEL
LIN {X 0,Y 503.357,Z 350.826,A -85,B 0,C 180,E1 -5838.218,E2 -5838.218} C_VEL
LIN {X 0,Y 503.094,Z 361.183,A -85,B 0,C 180,E1 -5839.13,E2 -5839.13} C_VEL
LIN {X 0,Y 502.774,Z 370.509,A -85,B 0,C 180,E1 -5840.14,E2 -5840.14} C_VEL
LIN {X 0,Y 502.513,Z 379.568,A -85,B 0,C 180,E1 -5841.353,E2 -5841.353} C_VEL
LIN {X 0,Y 502.349,Z 386.873,A -85,B 0,C 180,E1 -5842.565,E2 -5842.565} C_VEL
LIN {X 0,Y 502.235,Z 391.806,A -85,B 0,C 180,E1 -5843.572,E2 -5843.572} C_VEL
LIN {X 0,Y 502.179,Z 396.598,A -85,B 0,C 180,E1 -5844.781,E2 -5844.781} C_VEL
LIN {X 0,Y 502.166,Z 400.259,A -85,B 0,C 180,E1 -5845.987,E2 -5845.987} C_VEL
LIN {X 0,Y 502.122,Z 402.143,A -85,B 0,C 180,E1 -5846.791,E2 -5846.791} C_VEL
LIN {X 0,Y 502.121,Z 403.558,A -85,B 0,C 180,E1 -5847.594,E2 -5847.594} C_VEL
LIN {X 0,Y 501.995,Z 405.159,A -85,B 0,C 180,E1 -5849.198,E2 -5849.198} C_VEL
LIN {X 0,Y 501.992,Z 405.367,A -85,B 0,C 180,E1 -5850,E2 -5850} C_VEL
LIN {X 0,Y 501.996,Z 405.136,A -85,B 0,C 180,E1 -5850.802,E2 -5850.802} C_VEL
LIN {X 0,Y 502.036,Z 404.508,A -85,B 0,C 180,E1 -5851.605,E2 -5851.605} C_VEL
LIN {X 0,Y 502.121,Z 403.479,A -85,B 0,C 180,E1 -5852.407,E2 -5852.407} C_VEL
LIN {X 0,Y 502.123,Z 402.035,A -85,B 0,C 180,E1 -5853.21,E2 -5853.21} C_VEL
LIN {X 0,Y 502.117,Z 399.014,A -85,B 0,C 180,E1 -5854.415,E2 -5854.415} C_VEL
LIN {X 0,Y 502.222,Z 394.933,A -85,B 0,C 180,E1 -5855.622,E2 -5855.622} C_VEL
LIN {X 0,Y 502.324,Z 388.758,A -85,B 0,C 180,E1 -5857.012,E2 -5857.012} C_VEL
LIN {X 0,Y 502.44,Z 381.79,A -85,B 0,C 180,E1 -5858.243,E2 -5858.243} C_VEL
LIN {X 0,Y 502.682,Z 373.282,A -85,B 0,C 180,E1 -5859.455,E2 -5859.455} C_VEL
LIN {X 0,Y 502.948,Z 364.531,A -85,B 0,C 180,E1 -5860.466,E2 -5860.466} C_VEL
LIN {X 0,Y 503.287,Z 353.772,A -85,B 0,C 180,E1 -5861.478,E2 -5861.478} C_VEL
LIN {X 0,Y 503.556,Z 342.715,A -85,B 0,C 180,E1 -5862.319,E2 -5862.319} C_VEL
LIN {X 0,Y 503.883,Z 331.415,A -85,B 0,C 180,E1 -5862.998,E2 -5862.998} C_VEL
LIN {X 0,Y 504.256,Z 318.158,A -85,B 0,C 180,E1 -5863.603,E2 -5863.603} C_VEL
LIN {X 0,Y 504.217,Z 311.417,A -85,B 0,C 180,E1 -5863.848,E2 -5863.848} C_VEL
LIN {X 0,Y 502.648,Z 299.321,A -85,B 0,C 180,E1 -5864.215,E2 -5864.215} C_VEL
LIN {X 0,Y 502.331,Z 296.738,A -85,B 0,C 180,E1 -5864.276,E2 -5864.276} C_VEL
LIN {X 0,Y 502.449,Z 286.203,A -85,B 0,C 180,E1 -5867.502,E2 -5867.502} C_VEL
LIN {X 0,Y 502.59,Z 276.758,A -85,B 0,C 180,E1 -5870.462,E2 -5870.462} C_VEL
LIN {X 0,Y 502.715,Z 268.751,A -85,B 0,C 180,E1 -5873.045,E2 -5873.045} C_VEL
LIN {X 0,Y 502.969,Z 259.655,A -85,B 0,C 180,E1 -5876.114,E2 -5876.114} C_VEL
LIN {X 0,Y 503.158,Z 252.132,A -85,B 0,C 180,E1 -5878.809,E2 -5878.809} C_VEL
LIN {X 0,Y 503.656,Z 244.769,A -85,B 0,C 180,E1 -5881.658,E2 -5881.658} C_VEL
LIN {X 0,Y 504.065,Z 239.526,A -85,B 0,C 180,E1 -5883.898,E2 -5883.898} C_VEL
LIN {X 0,Y 504.22,Z 235.077,A -85,B 0,C 180,E1 -5886.057,E2 -5886.057} C_VEL
LIN {X 0,Y 503.88,Z 231.951,A -85,B 0,C 180,E1 -5887.858,E2 -5887.858} C_VEL
LIN {X 0,Y 503.386,Z 228.998,A -85,B 0,C 180,E1 -5889.958,E2 -5889.958} C_VEL
LIN {X 0,Y 502.933,Z 226.639,A -85,B 0,C 180,E1 -5892.215,E2 -5892.215} C_VEL
LIN {X 0,Y 502.774,Z 225.861,A -85,B 0,C 180,E1 -5893.374,E2 -5893.374} C_VEL
LIN {X 0,Y 502.783,Z 225.86,A -85,B 0,C 180,E1 -5895.66,E2 -5895.66} C_VEL
LIN {X 0,Y 502.822,Z 225.855,A -85,B 0,C 180,E1 -5899.005,E2 -5899.005} C_VEL
LIN {X 0,Y 502.797,Z 225.858,A -85,B 0,C 180,E1 -5902.046,E2 -5902.046} C_VEL
LIN {X 0,Y 502.794,Z 225.989,A -85,B 0,C 180,E1 -5903.055,E2 -5903.055} C_VEL
LIN {X 0,Y 502.94,Z 227.486,A -85,B 0,C 180,E1 -5905.534,E2 -5905.534} C_VEL
LIN {X 0,Y 502.786,Z 229.686,A -85,B 0,C 180,E1 -5908.503,E2 -5908.503} C_VEL
LIN {X 0,Y 502.711,Z 231.488,A -85,B 0,C 180,E1 -5910.705,E2 -5910.705} C_VEL
LIN {X 0,Y 502.59,Z 233.917,A -85,B 0,C 180,E1 -5913.503,E2 -5913.503} C_VEL
LIN {X 0,Y 502.493,Z 236.285,A -85,B 0,C 180,E1 -5916.071,E2 -5916.071} C_VEL
LIN {X 0,Y 502.395,Z 238.766,A -85,B 0,C 180,E1 -5918.672,E2 -5918.672} C_VEL
LIN {X 0,Y 502.381,Z 242.133,A -85,B 0,C 180,E1 -5922.075,E2 -5922.075} C_VEL
LIN {X 0,Y 502.323,Z 245.571,A -85,B 0,C 180,E1 -5925.414,E2 -5925.414} C_VEL
LIN {X 0,Y 502.257,Z 247.109,A -85,B 0,C 180,E1 -5926.857,E2 -5926.857} C_VEL
LIN {X 0,Y 504.635,Z 258.169,A -85,B 0,C 180,E1 -5927.248,E2 -5927.248} C_VEL
LIN {X 0,Y 504.426,Z 271.07,A -85,B 0,C 180,E1 -5927.769,E2 -5927.769} C_VEL
LIN {X 0,Y 504.14,Z 283.388,A -85,B 0,C 180,E1 -5928.44,E2 -5928.44} C_VEL
LIN {X 0,Y 503.719,Z 294.807,A -85,B 0,C 180,E1 -5929.245,E2 -5929.245} C_VEL
LIN {X 0,Y 503.354,Z 305.128,A -85,B 0,C 180,E1 -5930.152,E2 -5930.152} C_VEL
LIN {X 0,Y 503.106,Z 314.439,A -85,B 0,C 180,E1 -5931.161,E2 -5931.161} C_VEL
LIN {X 0,Y 502.746,Z 323.415,A -85,B 0,C 180,E1 -5932.368,E2 -5932.368} C_VEL
LIN {X 0,Y 502.589,Z 330.635,A -85,B 0,C 180,E1 -5933.577,E2 -5933.577} C_VEL
LIN {X 0,Y 502.392,Z 336.414,A -85,B 0,C 180,E1 -5934.783,E2 -5934.783} C_VEL
LIN {X 0,Y 502.274,Z 340.952,A -85,B 0,C 180,E1 -5935.988,E2 -5935.988} C_VEL
LIN {X 0,Y 502.298,Z 343.339,A -85,B 0,C 180,E1 -5936.792,E2 -5936.792} C_VEL
LIN {X 0,Y 502.15,Z 345.295,A -85,B 0,C 180,E1 -5937.594,E2 -5937.594} C_VEL
LIN {X 0,Y 502.049,Z 346.836,A -85,B 0,C 180,E1 -5938.396,E2 -5938.396} C_VEL
LIN {X 0,Y 502.012,Z 347.947,A -85,B 0,C 180,E1 -5939.198,E2 -5939.198} C_VEL
LIN {X 0,Y 502.004,Z 348.934,A -85,B 0,C 180,E1 -5940.802,E2 -5940.802} C_VEL
LIN {X 0,Y 502.038,Z 348.85,A -85,B 0,C 180,E1 -5941.604,E2 -5941.604} C_VEL
LIN {X 0,Y 502.129,Z 348.355,A -85,B 0,C 180,E1 -5942.407,E2 -5942.407} C_VEL
LIN {X 0,Y 502.191,Z 347.445,A -85,B 0,C 180,E1 -5943.209,E2 -5943.209} C_VEL
LIN {X 0,Y 502.192,Z 346.138,A -85,B 0,C 180,E1 -5944.013,E2 -5944.013} C_VEL
LIN {X 0,Y 502.17,Z 343.386,A -85,B 0,C 180,E1 -5945.219,E2 -5945.219} C_VEL
LIN {X 0,Y 502.239,Z 339.283,A -85,B 0,C 180,E1 -5946.518,E2 -5946.518} C_VEL
LIN {X 0,Y 502.423,Z 334.689,A -85,B 0,C 180,E1 -5947.637,E2 -5947.637} C_VEL
LIN {X 0,Y 502.598,Z 328.494,A -85,B 0,C 180,E1 -5948.848,E2 -5948.848} C_VEL
LIN {X 0,Y 502.796,Z 320.764,A -85,B 0,C 180,E1 -5950.063,E2 -5950.063} C_VEL
LIN {X 0,Y 503.118,Z 312.842,A -85,B 0,C 180,E1 -5951.074,E2 -5951.074} C_VEL
LIN {X 0,Y 503.339,Z 303.179,A -85,B 0,C 180,E1 -5952.09,E2 -5952.09} C_VEL
LIN {X 0,Y 503.718,Z 292.455,A -85,B 0,C 180,E1 -5953.002,E2 -5953.002} C_VEL
LIN {X 0,Y 504.098,Z 282.064,A -85,B 0,C 180,E1 -5953.71,E2 -5953.71} C_VEL
LIN {X 0,Y 504.363,Z 269.639,A -85,B 0,C 180,E1 -5954.372,E2 -5954.372} C_VEL
LIN {X 0,Y 504.493,Z 257.246,A -85,B 0,C 180,E1 -5954.864,E2 -5954.864} C_VEL
LIN {X 0,Y 502.139,Z 245.868,A -85,B 0,C 180,E1 -5955.265,E2 -5955.265} C_VEL
LIN {X 0,Y 502.209,Z 242.77,A -85,B 0,C 180,E1 -5957.931,E2 -5957.931} C_VEL
LIN {X 0,Y 502.176,Z 239.836,A -85,B 0,C 180,E1 -5960.48,E2 -5960.48} C_VEL
LIN {X 0,Y 502.18,Z 236.894,A -85,B 0,C 180,E1 -5963.07,E2 -5963.07} C_VEL
LIN {X 0,Y 502.281,Z 233.93,A -85,B 0,C 180,E1 -5965.706,E2 -5965.706} C_VEL
LIN {X 0,Y 502.296,Z 230.928,A -85,B 0,C 180,E1 -5968.406,E2 -5968.406} C_VEL
LIN {X 0,Y 502.321,Z 227.603,A -85,B 0,C 180,E1 -5971.41,E2 -5971.41} C_VEL
LIN {X 0,Y 502.356,Z 225.913,A -85,B 0,C 180,E1 -5973.067,E2 -5973.067} C_VEL
LIN {X 0,Y 502.686,Z 225.871,A -85,B 0,C 180,E1 -5975.959,E2 -5975.959} C_VEL
LIN {X 0,Y 502.797,Z 225.853,A -85,B 0,C 180,E1 -5978.977,E2 -5978.977} C_VEL
LIN {X 0,Y 502.808,Z 225.854,A -85,B 0,C 180,E1 -5982.199,E2 -5982.199} C_VEL
LIN {X 0,Y 502.79,Z 225.858,A -85,B 0,C 180,E1 -5985.47,E2 -5985.47} C_VEL
LIN {X 0,Y 502.758,Z 225.856,A -85,B 0,C 180,E1 -5988.349,E2 -5988.349} C_VEL
LIN {X 0,Y 502.78,Z 225.86,A -85,B 0,C 180,E1 -5991.022,E2 -5991.022} C_VEL
LIN {X 0,Y 502.753,Z 225.856,A -85,B 0,C 180,E1 -5991.833,E2 -5991.833} C_VEL
LIN {X 0,Y 502.093,Z 225.943,A -85,B 0,C 180,E1 -5992.502,E2 -5992.502} C_VEL
LIN {X 0,Y 499.238,Z 226.296,A -85,B 0,C 180,E1 -5993.587,E2 -5993.587} C_VEL
LIN {X 0,Y 496.837,Z 226.597,A -85,B 0,C 180,E1 -5994.462,E2 -5994.462} C_VEL
LIN {X 0,Y 495.83,Z 226.721,A -85,B 0,C 180,E1 -5995.138,E2 -5995.138} C_VEL
LIN {X 0,Y 495.761,Z 226.728,A -85,B 0,C 180,E1 -5995.367,E2 -5995.367} C_VEL
LIN {X 0,Y 495.758,Z 226.734,A -85,B 0,C 180,E1 -5998.364,E2 -5998.364} C_VEL
LIN {X 0,Y 495.759,Z 226.73,A -85,B 0,C 180,E1 -6001.514,E2 -6001.514} C_VEL
LIN {X 0,Y 495.766,Z 226.732,A -85,B 0,C 180,E1 -6003.93,E2 -6003.93} C_VEL
LIN {X 0,Y 495.764,Z 226.731,A -85,B 0,C 180,E1 -6007.139,E2 -6007.139} C_VEL
LIN {X 0,Y 495.775,Z 226.728,A -85,B 0,C 180,E1 -6010.11,E2 -6010.11} C_VEL
LIN {X 0,Y 495.766,Z 226.731,A -85,B 0,C 180,E1 -6012.68,E2 -6012.68} C_VEL
LIN {X 0,Y 495.79,Z 226.729,A -85,B 0,C 180,E1 -6015.217,E2 -6015.217} C_VEL
LIN {X 0,Y 495.855,Z 226.722,A -85,B 0,C 180,E1 -6018.555,E2 -6018.555} C_VEL
LIN {X 0,Y 495.817,Z 226.723,A -85,B 0,C 180,E1 -6021.851,E2 -6021.851} C_VEL
LIN {X 0,Y 495.817,Z 226.721,A -85,B 0,C 180,E1 -6025.121,E2 -6025.121} C_VEL
LIN {X 0,Y 495.978,Z 226.704,A -85,B 0,C 180,E1 -6027.563,E2 -6027.563} C_VEL
LIN {X 0,Y 495.979,Z 226.704,A -85,B 0,C 180,E1 -6030,E2 -6030} C_VEL
LIN {X 0,Y 495.991,Z 226.699,A -85,B 0,C 180,E1 -6032.436,E2 -6032.436} C_VEL
LIN {X 0,Y 495.614,Z 226.755,A -85,B 0,C 180,E1 -6035.697,E2 -6035.697} C_VEL
LIN {X 0,Y 495.521,Z 227.39,A -85,B 0,C 180,E1 -6036.106,E2 -6036.106} C_VEL
LIN {X 0,Y 495.477,Z 231.931,A -85,B 0,C 180,E1 -6038.154,E2 -6038.154} C_VEL
LIN {X 0,Y 495.475,Z 239.256,A -85,B 0,C 180,E1 -6041.454,E2 -6041.454} C_VEL
LIN {X 0,Y 495.423,Z 246.542,A -85,B 0,C 180,E1 -6044.794,E2 -6044.794} C_VEL
LIN {X 0,Y 495.333,Z 253.866,A -85,B 0,C 180,E1 -6048.189,E2 -6048.189} C_VEL
LIN {X 0,Y 495.223,Z 259.441,A -85,B 0,C 180,E1 -6050.781,E2 -6050.781} C_VEL
LIN {X 0,Y 495.172,Z 265.083,A -85,B 0,C 180,E1 -6053.416,E2 -6053.416} C_VEL
LIN {X 0,Y 495.212,Z 269.863,A -85,B 0,C 180,E1 -6055.649,E2 -6055.649} C_VEL
LIN {X 0,Y 496.742,Z 280.151,A -85,B 0,C 180,E1 -6056.014,E2 -6056.014} C_VEL
LIN {X 0,Y 496.549,Z 291.651,A -85,B 0,C 180,E1 -6056.534,E2 -6056.534} C_VEL
LIN {X 0,Y 496.318,Z 300.232,A -85,B 0,C 180,E1 -6057.058,E2 -6057.058} C_VEL
LIN {X 0,Y 496.109,Z 309.231,A -85,B 0,C 180,E1 -6057.757,E2 -6057.757} C_VEL
LIN {X 0,Y 495.907,Z 317.146,A -85,B 0,C 180,E1 -6058.518,E2 -6058.518} C_VEL
LIN {X 0,Y 495.685,Z 325.541,A -85,B 0,C 180,E1 -6059.518,E2 -6059.518} C_VEL
LIN {X 0,Y 495.488,Z 331.213,A -85,B 0,C 180,E1 -6060.365,E2 -6060.365} C_VEL
LIN {X 0,Y 495.314,Z 336.805,A -85,B 0,C 180,E1 -6061.407,E2 -6061.407} C_VEL
LIN {X 0,Y 495.192,Z 340.145,A -85,B 0,C 180,E1 -6062.155,E2 -6062.155} C_VEL
LIN {X 0,Y 495.115,Z 343.577,A -85,B 0,C 180,E1 -6063.124,E2 -6063.124} C_VEL
LIN {X 0,Y 495.093,Z 346.163,A -85,B 0,C 180,E1 -6064.088,E2 -6064.088} C_VEL
LIN {X 0,Y 494.96,Z 348.65,A -85,B 0,C 180,E1 -6065.603,E2 -6065.603} C_VEL
LIN {X 0,Y 494.91,Z 349.368,A -85,B 0,C 180,E1 -6066.614,E2 -6066.614} C_VEL
LIN {X 0,Y 494.916,Z 349.316,A -85,B 0,C 180,E1 -6067.634,E2 -6067.634} C_VEL
LIN {X 0,Y 494.955,Z 348.473,A -85,B 0,C 180,E1 -6068.665,E2 -6068.665} C_VEL
LIN {X 0,Y 495.047,Z 346.331,A -85,B 0,C 180,E1 -6069.948,E2 -6069.948} C_VEL
LIN {X 0,Y 495.143,Z 342.844,A -85,B 0,C 180,E1 -6071.212,E2 -6071.212} C_VEL
LIN {X 0,Y 495.269,Z 337.973,A -85,B 0,C 180,E1 -6072.447,E2 -6072.447} C_VEL
LIN {X 0,Y 495.373,Z 333.73,A -85,B 0,C 180,E1 -6073.295,E2 -6073.295} C_VEL
LIN {X 0,Y 495.539,Z 329.391,A -85,B 0,C 180,E1 -6074.023,E2 -6074.023} C_VEL
LIN {X 0,Y 495.715,Z 323.44,A -85,B 0,C 180,E1 -6074.856,E2 -6074.856} C_VEL
LIN {X 0,Y 495.961,Z 316.146,A -85,B 0,C 180,E1 -6075.693,E2 -6075.693} C_VEL
LIN {X 0,Y 496.155,Z 308.627,A -85,B 0,C 180,E1 -6076.401,E2 -6076.401} C_VEL
LIN {X 0,Y 496.402,Z 299.303,A -85,B 0,C 180,E1 -6077.111,E2 -6077.111} C_VEL
LIN {X 0,Y 496.64,Z 289.558,A -85,B 0,C 180,E1 -6077.675,E2 -6077.675} C_VEL
LIN {X 0,Y 496.729,Z 279.046,A -85,B 0,C 180,E1 -6078.122,E2 -6078.122} C_VEL
LIN {X 0,Y 495.18,Z 270.129,A -85,B 0,C 180,E1 -6078.44,E2 -6078.44} C_VEL
LIN {X 0,Y 495.254,Z 263.832,A -85,B 0,C 180,E1 -6081.362,E2 -6081.362} C_VEL
LIN {X 0,Y 495.241,Z 257.224,A -85,B 0,C 180,E1 -6084.42,E2 -6084.42} C_VEL
LIN {X 0,Y 495.386,Z 252.027,A -85,B 0,C 180,E1 -6086.828,E2 -6086.828} C_VEL
LIN {X 0,Y 495.364,Z 246.614,A -85,B 0,C 180,E1 -6089.286,E2 -6089.286} C_VEL
LIN {X 0,Y 495.369,Z 240.242,A -85,B 0,C 180,E1 -6092.083,E2 -6092.083} C_VEL
LIN {X 0,Y 495.451,Z 233.062,A -85,B 0,C 180,E1 -6095.21,E2 -6095.21} C_VEL
LIN {X 0,Y 495.514,Z 226.769,A -85,B 0,C 180,E1 -6097.923,E2 -6097.923} C_VEL
LIN {X 0,Y 495.754,Z 226.735,A -85,B 0,C 180,E1 -6100.109,E2 -6100.109} C_VEL
LIN {X 0,Y 495.767,Z 226.732,A -85,B 0,C 180,E1 -6102.681,E2 -6102.681} C_VEL
LIN {X 0,Y 495.792,Z 226.728,A -85,B 0,C 180,E1 -6105.217,E2 -6105.217} C_VEL
LIN {X 0,Y 495.855,Z 226.722,A -85,B 0,C 180,E1 -6108.555,E2 -6108.555} C_VEL
LIN {X 0,Y 495.876,Z 226.72,A -85,B 0,C 180,E1 -6111.852,E2 -6111.852} C_VEL
LIN {X 0,Y 495.84,Z 226.723,A -85,B 0,C 180,E1 -6115.121,E2 -6115.121} C_VEL
LIN {X 0,Y 495.996,Z 226.704,A -85,B 0,C 180,E1 -6117.564,E2 -6117.564} C_VEL
LIN {X 0,Y 495.986,Z 226.704,A -85,B 0,C 180,E1 -6120.812,E2 -6120.812} C_VEL
LIN {X 0,Y 495.997,Z 226.705,A -85,B 0,C 180,E1 -6122.436,E2 -6122.436} C_VEL
LIN {X 0,Y 495.885,Z 226.717,A -85,B 0,C 180,E1 -6125.694,E2 -6125.694} C_VEL
LIN {X 0,Y 495.842,Z 226.721,A -85,B 0,C 180,E1 -6128.97,E2 -6128.97} C_VEL
LIN {X 0,Y 495.832,Z 226.726,A -85,B 0,C 180,E1 -6132.035,E2 -6132.035} C_VEL
LIN {X 0,Y 495.827,Z 226.726,A -85,B 0,C 180,E1 -6135.452,E2 -6135.452} C_VEL
LIN {X 0,Y 495.781,Z 226.729,A -85,B 0,C 180,E1 -6138.237,E2 -6138.237} C_VEL
LIN {X 0,Y 495.777,Z 226.729,A -85,B 0,C 180,E1 -6140.756,E2 -6140.756} C_VEL
LIN {X 0,Y 495.743,Z 226.734,A -85,B 0,C 180,E1 -6143.388,E2 -6143.388} C_VEL
LIN {X 0,Y 495.808,Z 226.724,A -85,B 0,C 180,E1 -6146.745,E2 -6146.745} C_VEL
LIN {X 0,Y 495.768,Z 226.732,A -85,B 0,C 180,E1 -6149.746,E2 -6149.746} C_VEL
LIN {X 0,Y 495.768,Z 226.731,A -85,B 0,C 180,E1 -6152.594,E2 -6152.594} C_VEL
LIN {X 0,Y 495.749,Z 226.733,A -85,B 0,C 180,E1 -6155.538,E2 -6155.538} C_VEL
LIN {X 0,Y 495.765,Z 226.731,A -85,B 0,C 180,E1 -6158.768,E2 -6158.768} C_VEL
LIN {X 0,Y 495.758,Z 226.733,A -85,B 0,C 180,E1 -6161.781,E2 -6161.781} C_VEL
LIN {X 0,Y 495.739,Z 226.737,A -85,B 0,C 180,E1 -6165.141,E2 -6165.141} C_VEL
LIN {X 0,Y 495.758,Z 226.732,A -85,B 0,C 180,E1 -6168.219,E2 -6168.219} C_VEL
LIN {X 0,Y 495.758,Z 226.784,A -85,B 0,C 180,E1 -6170.586,E2 -6170.586} C_VEL
LIN {X 0,Y 497.028,Z 233.979,A -85,B 0,C 180,E1 -6173.567,E2 -6173.567} C_VEL
LIN {X 0,Y 497.111,Z 239.131,A -85,B 0,C 180,E1 -6175.562,E2 -6175.562} C_VEL
LIN {X 0,Y 496.682,Z 248.163,A -85,B 0,C 180,E1 -6178.904,E2 -6178.904} C_VEL
LIN {X 0,Y 496.274,Z 257.218,A -85,B 0,C 180,E1 -6182.139,E2 -6182.139} C_VEL
LIN {X 0,Y 496.009,Z 265.65,A -85,B 0,C 180,E1 -6185.07,E2 -6185.07} C_VEL
LIN {X 0,Y 495.772,Z 274.141,A -85,B 0,C 180,E1 -6187.935,E2 -6187.935} C_VEL
LIN {X 0,Y 495.554,Z 283.326,A -85,B 0,C 180,E1 -6190.962,E2 -6190.962} C_VEL
LIN {X 0,Y 495.36,Z 293.847,A -85,B 0,C 180,E1 -6194.362,E2 -6194.362} C_VEL
LIN {X 0,Y 495.28,Z 297.479,A -85,B 0,C 180,E1 -6195.517,E2 -6195.517} C_VEL
LIN {X 0,Y 497.21,Z 311.374,A -85,B 0,C 180,E1 -6195.927,E2 -6195.927} C_VEL
LIN {X 0,Y 497.505,Z 314.745,A -85,B 0,C 180,E1 -6196.053,E2 -6196.053} C_VEL
LIN {X 0,Y 497.168,Z 328.037,A -85,B 0,C 180,E1 -6196.616,E2 -6196.616} C_VEL
LIN {X 0,Y 496.752,Z 340.427,A -85,B 0,C 180,E1 -6197.33,E2 -6197.33} C_VEL
LIN {X 0,Y 496.32,Z 351.62,A -85,B 0,C 180,E1 -6198.152,E2 -6198.152} C_VEL
LIN {X 0,Y 496.031,Z 361.73,A -85,B 0,C 180,E1 -6199.076,E2 -6199.076} C_VEL
LIN {X 0,Y 495.662,Z 371.695,A -85,B 0,C 180,E1 -6200.204,E2 -6200.204} C_VEL
LIN {X 0,Y 495.434,Z 380.49,A -85,B 0,C 180,E1 -6201.434,E2 -6201.434} C_VEL
LIN {X 0,Y 495.266,Z 387.506,A -85,B 0,C 180,E1 -6202.663,E2 -6202.663} C_VEL
LIN {X 0,Y 495.112,Z 393.684,A -85,B 0,C 180,E1 -6204.029,E2 -6204.029} C_VEL
LIN {X 0,Y 495.037,Z 397.53,A -85,B 0,C 180,E1 -6205.114,E2 -6205.114} C_VEL
LIN {X 0,Y 495.058,Z 399.858,A -85,B 0,C 180,E1 -6205.93,E2 -6205.93} C_VEL
LIN {X 0,Y 495.045,Z 401.748,A -85,B 0,C 180,E1 -6206.745,E2 -6206.745} C_VEL
LIN {X 0,Y 495.054,Z 403.166,A -85,B 0,C 180,E1 -6207.559,E2 -6207.559} C_VEL
LIN {X 0,Y 494.915,Z 404.765,A -85,B 0,C 180,E1 -6209.186,E2 -6209.186} C_VEL
LIN {X 0,Y 494.909,Z 404.97,A -85,B 0,C 180,E1 -6210,E2 -6210} C_VEL
LIN {X 0,Y 494.915,Z 404.736,A -85,B 0,C 180,E1 -6210.814,E2 -6210.814} C_VEL
LIN {X 0,Y 495.054,Z 403.066,A -85,B 0,C 180,E1 -6212.441,E2 -6212.441} C_VEL
LIN {X 0,Y 495.046,Z 401.613,A -85,B 0,C 180,E1 -6213.256,E2 -6213.256} C_VEL
LIN {X 0,Y 495.02,Z 398.574,A -85,B 0,C 180,E1 -6214.479,E2 -6214.479} C_VEL
LIN {X 0,Y 495.135,Z 394.474,A -85,B 0,C 180,E1 -6215.702,E2 -6215.702} C_VEL
LIN {X 0,Y 495.254,Z 388.162,A -85,B 0,C 180,E1 -6217.133,E2 -6217.133} C_VEL
LIN {X 0,Y 495.365,Z 381.27,A -85,B 0,C 180,E1 -6218.362,E2 -6218.362} C_VEL
LIN {X 0,Y 495.608,Z 372.728,A -85,B 0,C 180,E1 -6219.592,E2 -6219.592} C_VEL
LIN {X 0,Y 495.901,Z 363.939,A -85,B 0,C 180,E1 -6220.617,E2 -6220.617} C_VEL
LIN {X 0,Y 496.252,Z 353.15,A -85,B 0,C 180,E1 -6221.643,E2 -6221.643} C_VEL
LIN {X 0,Y 496.57,Z 341.761,A -85,B 0,C 180,E1 -6222.516,E2 -6222.516} C_VEL
LIN {X 0,Y 496.925,Z 330.748,A -85,B 0,C 180,E1 -6223.183,E2 -6223.183} C_VEL
LIN {X 0,Y 497.341,Z 317.502,A -85,B 0,C 180,E1 -6223.796,E2 -6223.796} C_VEL
LIN {X 0,Y 497.212,Z 311.873,A -85,B 0,C 180,E1 -6224.008,E2 -6224.008} C_VEL
LIN {X 0,Y 495.43,Z 298.031,A -85,B 0,C 180,E1 -6224.441,E2 -6224.441} C_VEL
LIN {X 0,Y 495.221,Z 296.268,A -85,B 0,C 180,E1 -6224.485,E2 -6224.485} C_VEL
LIN {X 0,Y 495.371,Z 285.916,A -85,B 0,C 180,E1 -6227.719,E2 -6227.719} C_VEL
LIN {X 0,Y 495.527,Z 276.393,A -85,B 0,C 180,E1 -6230.767,E2 -6230.767} C_VEL
LIN {X 0,Y 495.68,Z 268.468,A -85,B 0,C 180,E1 -6233.391,E2 -6233.391} C_VEL
LIN {X 0,Y 495.955,Z 259.72,A -85,B 0,C 180,E1 -6236.422,E2 -6236.422} C_VEL
LIN {X 0,Y 496.199,Z 252.062,A -85,B 0,C 180,E1 -6239.252,E2 -6239.252} C_VEL
LIN {X 0,Y 496.675,Z 245.464,A -85,B 0,C 180,E1 -6241.896,E2 -6241.896} C_VEL
LIN {X 0,Y 497.168,Z 239.76,A -85,B 0,C 180,E1 -6244.433,E2 -6244.433} C_VEL
LIN {X 0,Y 497.21,Z 235.901,A -85,B 0,C 180,E1 -6246.418,E2 -6246.418} C_VEL
LIN {X 0,Y 496.821,Z 232.529,A -85,B 0,C 180,E1 -6248.494,E2 -6248.494} C_VEL
LIN {X 0,Y 496.327,Z 229.781,A -85,B 0,C 180,E1 -6250.645,E2 -6250.645} C_VEL
LIN {X 0,Y 495.894,Z 227.729,A -85,B 0,C 180,E1 -6252.866,E2 -6252.866} C_VEL
LIN {X 0,Y 495.741,Z 226.737,A -85,B 0,C 180,E1 -6254.859,E2 -6254.859} C_VEL
LIN {X 0,Y 495.76,Z 226.734,A -85,B 0,C 180,E1 -6258.219,E2 -6258.219} C_VEL
LIN {X 0,Y 495.754,Z 226.736,A -85,B 0,C 180,E1 -6261.409,E2 -6261.409} C_VEL
LIN {X 0,Y 495.872,Z 227.695,A -85,B 0,C 180,E1 -6263.888,E2 -6263.888} C_VEL
LIN {X 0,Y 495.902,Z 229.272,A -85,B 0,C 180,E1 -6266.447,E2 -6266.447} C_VEL
LIN {X 0,Y 495.744,Z 231.393,A -85,B 0,C 180,E1 -6269.312,E2 -6269.312} C_VEL
LIN {X 0,Y 495.592,Z 233.655,A -85,B 0,C 180,E1 -6272.097,E2 -6272.097} C_VEL
LIN {X 0,Y 495.508,Z 236.375,A -85,B 0,C 180,E1 -6275.196,E2 -6275.196} C_VEL
LIN {X 0,Y 495.353,Z 239.306,A -85,B 0,C 180,E1 -6278.353,E2 -6278.353} C_VEL
LIN {X 0,Y 495.333,Z 242.774,A -85,B 0,C 180,E1 -6281.922,E2 -6281.922} C_VEL
LIN {X 0,Y 495.267,Z 246.098,A -85,B 0,C 180,E1 -6285.201,E2 -6285.201} C_VEL
LIN {X 0,Y 495.189,Z 247.608,A -85,B 0,C 180,E1 -6286.64,E2 -6286.64} C_VEL
LIN {X 0,Y 497.749,Z 259.051,A -85,B 0,C 180,E1 -6287.072,E2 -6287.072} C_VEL
LIN {X 0,Y 497.523,Z 271.834,A -85,B 0,C 180,E1 -6287.604,E2 -6287.604} C_VEL
LIN {X 0,Y 497.227,Z 283.918,A -85,B 0,C 180,E1 -6288.277,E2 -6288.277} C_VEL
LIN {X 0,Y 496.766,Z 295.309,A -85,B 0,C 180,E1 -6289.093,E2 -6289.093} C_VEL
LIN {X 0,Y 496.38,Z 305.607,A -85,B 0,C 180,E1 -6290.012,E2 -6290.012} C_VEL
LIN {X 0,Y 496.121,Z 314.902,A -85,B 0,C 180,E1 -6291.035,E2 -6291.035} C_VEL
LIN {X 0,Y 495.733,Z 323.868,A -85,B 0,C 180,E1 -6292.26,E2 -6292.26} C_VEL
LIN {X 0,Y 495.554,Z 331.082,A -85,B 0,C 180,E1 -6293.485,E2 -6293.485} C_VEL
LIN {X 0,Y 495.346,Z 336.859,A -85,B 0,C 180,E1 -6294.709,E2 -6294.709} C_VEL
LIN {X 0,Y 495.217,Z 341.393,A -85,B 0,C 180,E1 -6295.931,E2 -6295.931} C_VEL
LIN {X 0,Y 495.243,Z 343.774,A -85,B 0,C 180,E1 -6296.746,E2 -6296.746} C_VEL
LIN {X 0,Y 495.087,Z 345.726,A -85,B 0,C 180,E1 -6297.559,E2 -6297.559} C_VEL
LIN {X 0,Y 494.976,Z 347.263,A -85,B 0,C 180,E1 -6298.373,E2 -6298.373} C_VEL
LIN {X 0,Y 494.931,Z 348.365,A -85,B 0,C 180,E1 -6299.186,E2 -6299.186} C_VEL
LIN {X 0,Y 494.923,Z 349.335,A -85,B 0,C 180,E1 -6300.814,E2 -6300.814} C_VEL
LIN {X 0,Y 494.965,Z 349.242,A -85,B 0,C 180,E1 -6301.627,E2 -6301.627} C_VEL
LIN {X 0,Y 495.064,Z 348.731,A -85,B 0,C 180,E1 -6302.441,E2 -6302.441} C_VEL
LIN {X 0,Y 495.108,Z 347.806,A -85,B 0,C 180,E1 -6303.255,E2 -6303.255} C_VEL
LIN {X 0,Y 495.124,Z 346.487,A -85,B 0,C 180,E1 -6304.07,E2 -6304.07} C_VEL
LIN {X 0,Y 495.112,Z 343.709,A -85,B 0,C 180,E1 -6305.294,E2 -6305.294} C_VEL
LIN {X 0,Y 495.202,Z 339.033,A -85,B 0,C 180,E1 -6306.754,E2 -6306.754} C_VEL
LIN {X 0,Y 495.365,Z 334.951,A -85,B 0,C 180,E1 -6307.746,E2 -6307.746} C_VEL
LIN {X 0,Y 495.568,Z 328.72,A -85,B 0,C 180,E1 -6308.975,E2 -6308.975} C_VEL
LIN {X 0,Y 495.784,Z 320.936,A -85,B 0,C 180,E1 -6310.207,E2 -6310.207} C_VEL
LIN {X 0,Y 496.128,Z 312.968,A -85,B 0,C 180,E1 -6311.232,E2 -6311.232} C_VEL
LIN {X 0,Y 496.388,Z 303.254,A -85,B 0,C 180,E1 -6312.262,E2 -6312.262} C_VEL
LIN {X 0,Y 496.782,Z 292.47,A -85,B 0,C 180,E1 -6313.187,E2 -6313.187} C_VEL
LIN {X 0,Y 497.253,Z 280.235,A -85,B 0,C 180,E1 -6314.007,E2 -6314.007} C_VEL
LIN {X 0,Y 497.512,Z 268.366,A -85,B 0,C 180,E1 -6314.626,E2 -6314.626} C_VEL
LIN {X 0,Y 497.613,Z 258.242,A -85,B 0,C 180,E1 -6315.029,E2 -6315.029} C_VEL
LIN {X 0,Y 495.083,Z 246.196,A -85,B 0,C 180,E1 -6315.461,E2 -6315.461} C_VEL
LIN {X 0,Y 495.119,Z 243.021,A -85,B 0,C 180,E1 -6318.197,E2 -6318.197} C_VEL
LIN {X 0,Y 495.095,Z 240.069,A -85,B 0,C 180,E1 -6320.786,E2 -6320.786} C_VEL
LIN {X 0,Y 495.116,Z 237.09,A -85,B 0,C 180,E1 -6323.419,E2 -6323.419} C_VEL
LIN {X 0,Y 495.24,Z 233.527,A -85,B 0,C 180,E1 -6326.614,E2 -6326.614} C_VEL
LIN {X 0,Y 495.265,Z 229.735,A -85,B 0,C 180,E1 -6330.046,E2 -6330.046} C_VEL
LIN {X 0,Y 495.256,Z 226.932,A -85,B 0,C 180,E1 -6332.632,E2 -6332.632} C_VEL
LIN {X 0,Y 495.608,Z 226.754,A -85,B 0,C 180,E1 -6335.55,E2 -6335.55} C_VEL
LIN {X 0,Y 495.751,Z 226.731,A -85,B 0,C 180,E1 -6338.766,E2 -6338.766} C_VEL
LIN {X 0,Y 495.755,Z 226.734,A -85,B 0,C 180,E1 -6341.782,E2 -6341.782} C_VEL
LIN {X 0,Y 495.741,Z 226.734,A -85,B 0,C 180,E1 -6345.141,E2 -6345.141} C_VEL
LIN {X 0,Y 495.738,Z 226.731,A -85,B 0,C 180,E1 -6348.217,E2 -6348.217} C_VEL
LIN {X 0,Y 495.737,Z 226.734,A -85,B 0,C 180,E1 -6351.236,E2 -6351.236} C_VEL
LIN {X 0,Y 495.73,Z 226.735,A -85,B 0,C 180,E1 -6354.46,E2 -6354.46} C_VEL
LIN {X 0,Y 495.761,Z 226.728,A -85,B 0,C 180,E1 -6355.367,E2 -6355.367} C_VEL
LIN {X 0,Y 495.125,Z 226.809,A -85,B 0,C 180,E1 -6356.045,E2 -6356.045} C_VEL
LIN {X 0,Y 492.268,Z 227.165,A -85,B 0,C 180,E1 -6357.145,E2 -6357.145} C_VEL
LIN {X 0,Y 489.829,Z 227.471,A -85,B 0,C 180,E1 -6358.031,E2 -6358.031} C_VEL
LIN {X 0,Y 488.777,Z 227.602,A -85,B 0,C 180,E1 -6358.716,E2 -6358.716} C_VEL
LIN {X 0,Y 488.69,Z 227.61,A -85,B 0,C 180,E1 -6358.948,E2 -6358.948} C_VEL
LIN {X 0,Y 488.717,Z 227.608,A -85,B 0,C 180,E1 -6361.669,E2 -6361.669} C_VEL
LIN {X 0,Y 488.72,Z 227.607,A -85,B 0,C 180,E1 -6364.442,E2 -6364.442} C_VEL
LIN {X 0,Y 488.726,Z 227.608,A -85,B 0,C 180,E1 -6367.153,E2 -6367.153} C_VEL
LIN {X 0,Y 488.729,Z 227.608,A -85,B 0,C 180,E1 -6369.81,E2 -6369.81} C_VEL
LIN {X 0,Y 488.717,Z 227.607,A -85,B 0,C 180,E1 -6372.423,E2 -6372.423} C_VEL
LIN {X 0,Y 488.764,Z 227.604,A -85,B 0,C 180,E1 -6374.999,E2 -6374.999} C_VEL
LIN {X 0,Y 488.809,Z 227.599,A -85,B 0,C 180,E1 -6378.387,E2 -6378.387} C_VEL
LIN {X 0,Y 488.765,Z 227.601,A -85,B 0,C 180,E1 -6381.733,E2 -6381.733} C_VEL
LIN {X 0,Y 488.806,Z 227.599,A -85,B 0,C 180,E1 -6384.223,E2 -6384.223} C_VEL
LIN {X 0,Y 488.944,Z 227.58,A -85,B 0,C 180,E1 -6387.528,E2 -6387.528} C_VEL
LIN {X 0,Y 488.948,Z 227.579,A -85,B 0,C 180,E1 -6390,E2 -6390} C_VEL
LIN {X 0,Y 488.957,Z 227.575,A -85,B 0,C 180,E1 -6392.471,E2 -6392.471} C_VEL
LIN {X 0,Y 488.705,Z 227.612,A -85,B 0,C 180,E1 -6394.95,E2 -6394.95} C_VEL
LIN {X 0,Y 488.505,Z 227.748,A -85,B 0,C 180,E1 -6395.883,E2 -6395.883} C_VEL
LIN {X 0,Y 488.428,Z 233.041,A -85,B 0,C 180,E1 -6398.273,E2 -6398.273} C_VEL
LIN {X 0,Y 488.441,Z 241.056,A -85,B 0,C 180,E1 -6401.921,E2 -6401.921} C_VEL
LIN {X 0,Y 488.356,Z 248.543,A -85,B 0,C 180,E1 -6405.375,E2 -6405.375} C_VEL
LIN {X 0,Y 488.244,Z 255.179,A -85,B 0,C 180,E1 -6408.462,E2 -6408.462} C_VEL
LIN {X 0,Y 488.161,Z 260.81,A -85,B 0,C 180,E1 -6411.095,E2 -6411.095} C_VEL
LIN {X 0,Y 488.089,Z 266.548,A -85,B 0,C 180,E1 -6413.777,E2 -6413.777} C_VEL
LIN {X 0,Y 488.152,Z 270.199,A -85,B 0,C 180,E1 -6415.491,E2 -6415.491} C_VEL
LIN {X 0,Y 489.741,Z 280.072,A -85,B 0,C 180,E1 -6415.842,E2 -6415.842} C_VEL
LIN {X 0,Y 489.602,Z 291.66,A -85,B 0,C 180,E1 -6416.365,E2 -6416.365} C_VEL
LIN {X 0,Y 489.323,Z 301.37,A -85,B 0,C 180,E1 -6416.975,E2 -6416.975} C_VEL
LIN {X 0,Y 489.121,Z 309.371,A -85,B 0,C 180,E1 -6417.606,E2 -6417.606} C_VEL
LIN {X 0,Y 488.928,Z 316.749,A -85,B 0,C 180,E1 -6418.317,E2 -6418.317} C_VEL
LIN {X 0,Y 488.698,Z 323.585,A -85,B 0,C 180,E1 -6419.114,E2 -6419.114} C_VEL
LIN {X 0,Y 488.475,Z 329.837,A -85,B 0,C 180,E1 -6419.998,E2 -6419.998} C_VEL
LIN {X 0,Y 488.279,Z 336.644,A -85,B 0,C 180,E1 -6421.209,E2 -6421.209} C_VEL
LIN {X 0,Y 488.121,Z 340.896,A -85,B 0,C 180,E1 -6422.19,E2 -6422.19} C_VEL
LIN {X 0,Y 488.038,Z 344.747,A -85,B 0,C 180,E1 -6423.36,E2 -6423.36} C_VEL
LIN {X 0,Y 488.007,Z 346.786,A -85,B 0,C 180,E1 -6424.17,E2 -6424.17} C_VEL
LIN {X 0,Y 487.909,Z 348.569,A -85,B 0,C 180,E1 -6425.182,E2 -6425.182} C_VEL
LIN {X 0,Y 487.854,Z 349.598,A -85,B 0,C 180,E1 -6426.222,E2 -6426.222} C_VEL
LIN {X 0,Y 487.839,Z 349.718,A -85,B 0,C 180,E1 -6427.594,E2 -6427.594} C_VEL
LIN {X 0,Y 487.882,Z 348.583,A -85,B 0,C 180,E1 -6428.933,E2 -6428.933} C_VEL
LIN {X 0,Y 488.041,Z 345.733,A -85,B 0,C 180,E1 -6430.393,E2 -6430.393} C_VEL
LIN {X 0,Y 488.132,Z 342.334,A -85,B 0,C 180,E1 -6431.523,E2 -6431.523} C_VEL
LIN {X 0,Y 488.22,Z 338.131,A -85,B 0,C 180,E1 -6432.577,E2 -6432.577} C_VEL
LIN {X 0,Y 488.394,Z 332.464,A -85,B 0,C 180,E1 -6433.687,E2 -6433.687} C_VEL
LIN {X 0,Y 488.647,Z 325.085,A -85,B 0,C 180,E1 -6434.809,E2 -6434.809} C_VEL
LIN {X 0,Y 488.923,Z 317.251,A -85,B 0,C 180,E1 -6435.741,E2 -6435.741} C_VEL
LIN {X 0,Y 489.139,Z 309.466,A -85,B 0,C 180,E1 -6436.495,E2 -6436.495} C_VEL
LIN {X 0,Y 489.388,Z 300.971,A -85,B 0,C 180,E1 -6437.161,E2 -6437.161} C_VEL
LIN {X 0,Y 489.668,Z 290.339,A -85,B 0,C 180,E1 -6437.808,E2 -6437.808} C_VEL
LIN {X 0,Y 489.784,Z 280.029,A -85,B 0,C 180,E1 -6438.259,E2 -6438.259} C_VEL
LIN {X 0,Y 488.12,Z 270.481,A -85,B 0,C 180,E1 -6438.609,E2 -6438.609} C_VEL
LIN {X 0,Y 488.194,Z 263.722,A -85,B 0,C 180,E1 -6441.755,E2 -6441.755} C_VEL
LIN {X 0,Y 488.242,Z 256.456,A -85,B 0,C 180,E1 -6445.134,E2 -6445.134} C_VEL
LIN {X 0,Y 488.321,Z 251.788,A -85,B 0,C 180,E1 -6447.336,E2 -6447.336} C_VEL
LIN {X 0,Y 488.326,Z 245.233,A -85,B 0,C 180,E1 -6450.229,E2 -6450.229} C_VEL
LIN {X 0,Y 488.33,Z 238.592,A -85,B 0,C 180,E1 -6453.164,E2 -6453.164} C_VEL
LIN {X 0,Y 488.413,Z 231.471,A -85,B 0,C 180,E1 -6456.24,E2 -6456.24} C_VEL
LIN {X 0,Y 488.475,Z 227.646,A -85,B 0,C 180,E1 -6457.921,E2 -6457.921} C_VEL
LIN {X 0,Y 488.698,Z 227.615,A -85,B 0,C 180,E1 -6459.809,E2 -6459.809} C_VEL
LIN {X 0,Y 488.717,Z 227.612,A -85,B 0,C 180,E1 -6462.423,E2 -6462.423} C_VEL
LIN {X 0,Y 488.765,Z 227.604,A -85,B 0,C 180,E1 -6465,E2 -6465} C_VEL
LIN {X 0,Y 488.809,Z 227.601,A -85,B 0,C 180,E1 -6468.387,E2 -6468.387} C_VEL
LIN {X 0,Y 488.821,Z 227.599,A -85,B 0,C 180,E1 -6471.734,E2 -6471.734} C_VEL
LIN {X 0,Y 488.809,Z 227.599,A -85,B 0,C 180,E1 -6475.051,E2 -6475.051} C_VEL
LIN {X 0,Y 488.964,Z 227.58,A -85,B 0,C 180,E1 -6477.529,E2 -6477.529} C_VEL
LIN {X 0,Y 488.937,Z 227.582,A -85,B 0,C 180,E1 -6480.824,E2 -6480.824} C_VEL
LIN {X 0,Y 488.964,Z 227.581,A -85,B 0,C 180,E1 -6482.471,E2 -6482.471} C_VEL
LIN {X 0,Y 488.842,Z 227.595,A -85,B 0,C 180,E1 -6485.776,E2 -6485.776} C_VEL
LIN {X 0,Y 488.819,Z 227.598,A -85,B 0,C 180,E1 -6488.266,E2 -6488.266} C_VEL
LIN {X 0,Y 488.809,Z 227.597,A -85,B 0,C 180,E1 -6491.612,E2 -6491.612} C_VEL
LIN {X 0,Y 488.765,Z 227.603,A -85,B 0,C 180,E1 -6495,E2 -6495} C_VEL
LIN {X 0,Y 488.75,Z 227.604,A -85,B 0,C 180,E1 -6498.442,E2 -6498.442} C_VEL
LIN {X 0,Y 488.709,Z 227.61,A -85,B 0,C 180,E1 -6501.071,E2 -6501.071} C_VEL
LIN {X 0,Y 488.675,Z 227.616,A -85,B 0,C 180,E1 -6503.746,E2 -6503.746} C_VEL
LIN {X 0,Y 488.75,Z 227.603,A -85,B 0,C 180,E1 -6506.933,E2 -6506.933} C_VEL
LIN {X 0,Y 488.725,Z 227.607,A -85,B 0,C 180,E1 -6509.27,E2 -6509.27} C_VEL
LIN {X 0,Y 488.704,Z 227.612,A -85,B 0,C 180,E1 -6512.147,E2 -6512.147} C_VEL
LIN {X 0,Y 488.717,Z 227.608,A -85,B 0,C 180,E1 -6515.115,E2 -6515.115} C_VEL
LIN {X 0,Y 488.682,Z 227.616,A -85,B 0,C 180,E1 -6518.2,E2 -6518.2} C_VEL
LIN {X 0,Y 488.72,Z 227.609,A -85,B 0,C 180,E1 -6520.345,E2 -6520.345} C_VEL
LIN {X 0,Y 488.686,Z 227.613,A -85,B 0,C 180,E1 -6523.655,E2 -6523.655} C_VEL
LIN {X 0,Y 488.686,Z 227.616,A -85,B 0,C 180,E1 -6526.345,E2 -6526.345} C_VEL
LIN {X 0,Y 488.735,Z 227.607,A -85,B 0,C 180,E1 -6529.677,E2 -6529.677} C_VEL
LIN {X 0,Y 488.742,Z 227.69,A -85,B 0,C 180,E1 -6530.349,E2 -6530.349} C_VEL
LIN {X 0,Y 490.005,Z 235.013,A -85,B 0,C 180,E1 -6533.436,E2 -6533.436} C_VEL
LIN {X 0,Y 490.14,Z 240.254,A -85,B 0,C 180,E1 -6535.502,E2 -6535.502} C_VEL
LIN {X 0,Y 489.688,Z 249.265,A -85,B 0,C 180,E1 -6538.891,E2 -6538.891} C_VEL
LIN {X 0,Y 489.29,Z 257.023,A -85,B 0,C 180,E1 -6541.706,E2 -6541.706} C_VEL
LIN {X 0,Y 488.968,Z 266.043,A -85,B 0,C 180,E1 -6544.892,E2 -6544.892} C_VEL
LIN {X 0,Y 488.696,Z 275.203,A -85,B 0,C 180,E1 -6548.043,E2 -6548.043} C_VEL
LIN {X 0,Y 488.471,Z 284.359,A -85,B 0,C 180,E1 -6551.112,E2 -6551.112} C_VEL
LIN {X 0,Y 488.254,Z 295.181,A -85,B 0,C 180,E1 -6554.668,E2 -6554.668} C_VEL
LIN {X 0,Y 488.198,Z 297.128,A -85,B 0,C 180,E1 -6555.302,E2 -6555.302} C_VEL
LIN {X 0,Y 490.198,Z 311.607,A -85,B 0,C 180,E1 -6555.748,E2 -6555.748} C_VEL
LIN {X 0,Y 490.559,Z 315.652,A -85,B 0,C 180,E1 -6555.904,E2 -6555.904} C_VEL
LIN {X 0,Y 490.249,Z 327.522,A -85,B 0,C 180,E1 -6556.423,E2 -6556.423} C_VEL
LIN {X 0,Y 489.826,Z 338.857,A -85,B 0,C 180,E1 -6557.077,E2 -6557.077} C_VEL
LIN {X 0,Y 489.336,Z 351.128,A -85,B 0,C 180,E1 -6557.98,E2 -6557.98} C_VEL
LIN {X 0,Y 489.044,Z 361.265,A -85,B 0,C 180,E1 -6558.918,E2 -6558.918} C_VEL
LIN {X 0,Y 488.613,Z 371.241,A -85,B 0,C 180,E1 -6560.061,E2 -6560.061} C_VEL
LIN {X 0,Y 488.349,Z 380.051,A -85,B 0,C 180,E1 -6561.309,E2 -6561.309} C_VEL
LIN {X 0,Y 488.19,Z 387.085,A -85,B 0,C 180,E1 -6562.556,E2 -6562.556} C_VEL
LIN {X 0,Y 488.021,Z 392.691,A -85,B 0,C 180,E1 -6563.794,E2 -6563.794} C_VEL
LIN {X 0,Y 487.968,Z 397.128,A -85,B 0,C 180,E1 -6565.043,E2 -6565.043} C_VEL
LIN {X 0,Y 487.952,Z 399.459,A -85,B 0,C 180,E1 -6565.87,E2 -6565.87} C_VEL
LIN {X 0,Y 487.969,Z 401.353,A -85,B 0,C 180,E1 -6566.697,E2 -6566.697} C_VEL
LIN {X 0,Y 487.959,Z 402.773,A -85,B 0,C 180,E1 -6567.524,E2 -6567.524} C_VEL
LIN {X 0,Y 487.893,Z 403.77,A -85,B 0,C 180,E1 -6568.349,E2 -6568.349} C_VEL
LIN {X 0,Y 487.838,Z 404.371,A -85,B 0,C 180,E1 -6569.175,E2 -6569.175} C_VEL
LIN {X 0,Y 487.829,Z 404.574,A -85,B 0,C 180,E1 -6570,E2 -6570} C_VEL
LIN {X 0,Y 487.838,Z 404.336,A -85,B 0,C 180,E1 -6570.826,E2 -6570.826} C_VEL
LIN {X 0,Y 487.893,Z 403.693,A -85,B 0,C 180,E1 -6571.651,E2 -6571.651} C_VEL
LIN {X 0,Y 487.959,Z 402.651,A -85,B 0,C 180,E1 -6572.477,E2 -6572.477} C_VEL
LIN {X 0,Y 487.97,Z 401.191,A -85,B 0,C 180,E1 -6573.303,E2 -6573.303} C_VEL
LIN {X 0,Y 487.93,Z 398.135,A -85,B 0,C 180,E1 -6574.544,E2 -6574.544} C_VEL
LIN {X 0,Y 488.028,Z 394.014,A -85,B 0,C 180,E1 -6575.786,E2 -6575.786} C_VEL
LIN {X 0,Y 488.181,Z 387.67,A -85,B 0,C 180,E1 -6577.237,E2 -6577.237} C_VEL
LIN {X 0,Y 488.313,Z 380.758,A -85,B 0,C 180,E1 -6578.484,E2 -6578.484} C_VEL
LIN {X 0,Y 488.552,Z 372.187,A -85,B 0,C 180,E1 -6579.732,E2 -6579.732} C_VEL
LIN {X 0,Y 488.857,Z 363.372,A -85,B 0,C 180,E1 -6580.772,E2 -6580.772} C_VEL
LIN {X 0,Y 489.185,Z 352.729,A -85,B 0,C 180,E1 -6581.798,E2 -6581.798} C_VEL
LIN {X 0,Y 489.603,Z 340.836,A -85,B 0,C 180,E1 -6582.719,E2 -6582.719} C_VEL
LIN {X 0,Y 490.08,Z 328.203,A -85,B 0,C 180,E1 -6583.476,E2 -6583.476} C_VEL
LIN {X 0,Y 490.505,Z 315.715,A -85,B 0,C 180,E1 -6584.045,E2 -6584.045} C_VEL
LIN {X 0,Y 489.021,Z 302.217,A -85,B 0,C 180,E1 -6584.527,E2 -6584.527} C_VEL
LIN {X 0,Y 488.176,Z 295.725,A -85,B 0,C 180,E1 -6584.726,E2 -6584.726} C_VEL
LIN {X 0,Y 488.335,Z 284.774,A -85,B 0,C 180,E1 -6588.221,E2 -6588.221} C_VEL
LIN {X 0,Y 488.539,Z 274.738,A -85,B 0,C 180,E1 -6591.521,E2 -6591.521} C_VEL
LIN {X 0,Y 488.714,Z 265.624,A -85,B 0,C 180,E1 -6594.648,E2 -6594.648} C_VEL
LIN {X 0,Y 489.007,Z 258.072,A -85,B 0,C 180,E1 -6597.381,E2 -6597.381} C_VEL
LIN {X 0,Y 489.4,Z 250.067,A -85,B 0,C 180,E1 -6600.5,E2 -6600.5} C_VEL
LIN {X 0,Y 489.933,Z 244.145,A -85,B 0,C 180,E1 -6603.032,E2 -6603.032} C_VEL
LIN {X 0,Y 490.31,Z 239.599,A -85,B 0,C 180,E1 -6605.212,E2 -6605.212} C_VEL
LIN {X 0,Y 490.167,Z 236.348,A -85,B 0,C 180,E1 -6607.028,E2 -6607.028} C_VEL
LIN {X 0,Y 489.711,Z 233.119,A -85,B 0,C 180,E1 -6609.197,E2 -6609.197} C_VEL
LIN {X 0,Y 489.212,Z 230.329,A -85,B 0,C 180,E1 -6611.666,E2 -6611.666} C_VEL
LIN {X 0,Y 488.807,Z 228.161,A -85,B 0,C 180,E1 -6614.791,E2 -6614.791} C_VEL
LIN {X 0,Y 488.713,Z 227.612,A -85,B 0,C 180,E1 -6617.174,E2 -6617.174} C_VEL
LIN {X 0,Y 488.737,Z 227.609,A -85,B 0,C 180,E1 -6619.677,E2 -6619.677} C_VEL
LIN {X 0,Y 488.808,Z 228.229,A -85,B 0,C 180,E1 -6622.259,E2 -6622.259} C_VEL
LIN {X 0,Y 488.953,Z 229.554,A -85,B 0,C 180,E1 -6625.015,E2 -6625.015} C_VEL
LIN {X 0,Y 488.795,Z 231.522,A -85,B 0,C 180,E1 -6628.03,E2 -6628.03} C_VEL
LIN {X 0,Y 488.636,Z 233.553,A -85,B 0,C 180,E1 -6630.724,E2 -6630.724} C_VEL
LIN {X 0,Y 488.509,Z 235.846,A -85,B 0,C 180,E1 -6633.514,E2 -6633.514} C_VEL
LIN {X 0,Y 488.391,Z 238.239,A -85,B 0,C 180,E1 -6636.239,E2 -6636.239} C_VEL
LIN {X 0,Y 488.293,Z 241.087,A -85,B 0,C 180,E1 -6639.318,E2 -6639.318} C_VEL
LIN {X 0,Y 488.244,Z 244.058,A -85,B 0,C 180,E1 -6642.405,E2 -6642.405} C_VEL
LIN {X 0,Y 488.214,Z 246.638,A -85,B 0,C 180,E1 -6644.982,E2 -6644.982} C_VEL
LIN {X 0,Y 488.142,Z 248.122,A -85,B 0,C 180,E1 -6646.417,E2 -6646.417} C_VEL
LIN {X 0,Y 490.878,Z 260.027,A -85,B 0,C 180,E1 -6646.889,E2 -6646.889} C_VEL
LIN {X 0,Y 490.623,Z 272.707,A -85,B 0,C 180,E1 -6647.433,E2 -6647.433} C_VEL
LIN {X 0,Y 490.318,Z 284.558,A -85,B 0,C 180,E1 -6648.109,E2 -6648.109} C_VEL
LIN {X 0,Y 489.835,Z 295.879,A -85,B 0,C 180,E1 -6648.936,E2 -6648.936} C_VEL
LIN {X 0,Y 489.427,Z 306.13,A -85,B 0,C 180,E1 -6649.869,E2 -6649.869} C_VEL
LIN {X 0,Y 489.138,Z 315.39,A -85,B 0,C 180,E1 -6650.906,E2 -6650.906} C_VEL
LIN {X 0,Y 488.723,Z 324.337,A -85,B 0,C 180,E1 -6652.148,E2 -6652.148} C_VEL
LIN {X 0,Y 488.522,Z 331.547,A -85,B 0,C 180,E1 -6653.391,E2 -6653.391} C_VEL
LIN {X 0,Y 488.303,Z 337.315,A -85,B 0,C 180,E1 -6654.632,E2 -6654.632} C_VEL
LIN {X 0,Y 488.162,Z 341.84,A -85,B 0,C 180,E1 -6655.872,E2 -6655.872} C_VEL
LIN {X 0,Y 488.189,Z 344.214,A -85,B 0,C 180,E1 -6656.699,E2 -6656.699} C_VEL
LIN {X 0,Y 488.027,Z 346.161,A -85,B 0,C 180,E1 -6657.524,E2 -6657.524} C_VEL
LIN {X 0,Y 487.905,Z 347.693,A -85,B 0,C 180,E1 -6658.349,E2 -6658.349} C_VEL
LIN {X 0,Y 487.853,Z 348.784,A -85,B 0,C 180,E1 -6659.175,E2 -6659.175} C_VEL
LIN {X 0,Y 487.846,Z 349.737,A -85,B 0,C 180,E1 -6660.826,E2 -6660.826} C_VEL
LIN {X 0,Y 487.895,Z 349.635,A -85,B 0,C 180,E1 -6661.651,E2 -6661.651} C_VEL
LIN {X 0,Y 488.001,Z 349.106,A -85,B 0,C 180,E1 -6662.476,E2 -6662.476} C_VEL
LIN {X 0,Y 488.029,Z 348.168,A -85,B 0,C 180,E1 -6663.302,E2 -6663.302} C_VEL
LIN {X 0,Y 488.058,Z 346.836,A -85,B 0,C 180,E1 -6664.129,E2 -6664.129} C_VEL
LIN {X 0,Y 488.056,Z 344.031,A -85,B 0,C 180,E1 -6665.371,E2 -6665.371} C_VEL
LIN {X 0,Y 488.125,Z 339.622,A -85,B 0,C 180,E1 -6666.77,E2 -6666.77} C_VEL
LIN {X 0,Y 488.331,Z 335.211,A -85,B 0,C 180,E1 -6667.858,E2 -6667.858} C_VEL
LIN {X 0,Y 488.517,Z 328.946,A -85,B 0,C 180,E1 -6669.106,E2 -6669.106} C_VEL
LIN {X 0,Y 488.787,Z 321.104,A -85,B 0,C 180,E1 -6670.354,E2 -6670.354} C_VEL
LIN {X 0,Y 489.198,Z 311.303,A -85,B 0,C 180,E1 -6671.603,E2 -6671.603} C_VEL
LIN {X 0,Y 489.537,Z 301.126,A -85,B 0,C 180,E1 -6672.646,E2 -6672.646} C_VEL
LIN {X 0,Y 489.958,Z 289.633,A -85,B 0,C 180,E1 -6673.585,E2 -6673.585} C_VEL
LIN {X 0,Y 490.445,Z 278.398,A -85,B 0,C 180,E1 -6674.311,E2 -6674.311} C_VEL
LIN {X 0,Y 490.671,Z 267.009,A -85,B 0,C 180,E1 -6674.888,E2 -6674.888} C_VEL
LIN {X 0,Y 490.585,Z 258.526,A -85,B 0,C 180,E1 -6675.226,E2 -6675.226} C_VEL
LIN {X 0,Y 487.982,Z 246.511,A -85,B 0,C 180,E1 -6675.667,E2 -6675.667} C_VEL
LIN {X 0,Y 488.029,Z 243.284,A -85,B 0,C 180,E1 -6678.471,E2 -6678.471} C_VEL
LIN {X 0,Y 488.011,Z 240.292,A -85,B 0,C 180,E1 -6681.102,E2 -6681.102} C_VEL
LIN {X 0,Y 488.053,Z 237.282,A -85,B 0,C 180,E1 -6683.779,E2 -6683.779} C_VEL
LIN {X 0,Y 488.173,Z 233.926,A -85,B 0,C 180,E1 -6686.799,E2 -6686.799} C_VEL
LIN {X 0,Y 488.178,Z 231.183,A -85,B 0,C 180,E1 -6689.306,E2 -6689.306} C_VEL
LIN {X 0,Y 488.189,Z 228.06,A -85,B 0,C 180,E1 -6692.185,E2 -6692.185} C_VEL
LIN {X 0,Y 488.322,Z 227.661,A -85,B 0,C 180,E1 -6693.41,E2 -6693.41} C_VEL
LIN {X 0,Y 488.604,Z 227.623,A -85,B 0,C 180,E1 -6696.341,E2 -6696.341} C_VEL
LIN {X 0,Y 488.699,Z 227.609,A -85,B 0,C 180,E1 -6699.255,E2 -6699.255} C_VEL
LIN {X 0,Y 488.702,Z 227.613,A -85,B 0,C 180,E1 -6701.598,E2 -6701.598} C_VEL
LIN {X 0,Y 488.705,Z 227.608,A -85,B 0,C 180,E1 -6704.803,E2 -6704.803} C_VEL
LIN {X 0,Y 488.67,Z 227.615,A -85,B 0,C 180,E1 -6707.472,E2 -6707.472} C_VEL
LIN {X 0,Y 488.707,Z 227.608,A -85,B 0,C 180,E1 -6709.674,E2 -6709.674} C_VEL
LIN {X 0,Y 488.649,Z 227.621,A -85,B 0,C 180,E1 -6712.838,E2 -6712.838} C_VEL
LIN {X 0,Y 488.719,Z 227.605,A -85,B 0,C 180,E1 -6715.886,E2 -6715.886} C_VEL
LIN {X 0,Y 488.69,Z 227.61,A -85,B 0,C 180,E1 -6718.948,E2 -6718.948} C_VEL
LIN {X 0,Y 488.018,Z 227.694,A -85,B 0,C 180,E1 -6719.637,E2 -6719.637} C_VEL
LIN {X 0,Y 485.16,Z 228.051,A -85,B 0,C 180,E1 -6720.754,E2 -6720.754} C_VEL
LIN {X 0,Y 482.76,Z 228.351,A -85,B 0,C 180,E1 -6721.655,E2 -6721.655} C_VEL
LIN {X 0,Y 481.751,Z 228.478,A -85,B 0,C 180,E1 -6722.351,E2 -6722.351} C_VEL
LIN {X 0,Y 481.68,Z 228.484,A -85,B 0,C 180,E1 -6722.587,E2 -6722.587} C_VEL
LIN {X 0,Y 481.662,Z 228.49,A -85,B 0,C 180,E1 -6725.886,E2 -6725.886} C_VEL
LIN {X 0,Y 481.707,Z 228.482,A -85,B 0,C 180,E1 -6729.027,E2 -6729.027} C_VEL
LIN {X 0,Y 481.695,Z 228.482,A -85,B 0,C 180,E1 -6732.158,E2 -6732.158} C_VEL
LIN {X 0,Y 481.746,Z 228.479,A -85,B 0,C 180,E1 -6734.776,E2 -6734.776} C_VEL
LIN {X 0,Y 481.755,Z 228.476,A -85,B 0,C 180,E1 -6738.215,E2 -6738.215} C_VEL
LIN {X 0,Y 481.724,Z 228.478,A -85,B 0,C 180,E1 -6741.611,E2 -6741.611} C_VEL
LIN {X 0,Y 481.767,Z 228.477,A -85,B 0,C 180,E1 -6744.139,E2 -6744.139} C_VEL
LIN {X 0,Y 481.909,Z 228.456,A -85,B 0,C 180,E1 -6747.492,E2 -6747.492} C_VEL
LIN {X 0,Y 481.918,Z 228.455,A -85,B 0,C 180,E1 -6750,E2 -6750} C_VEL
LIN {X 0,Y 481.923,Z 228.451,A -85,B 0,C 180,E1 -6752.507,E2 -6752.507} C_VEL
LIN {X 0,Y 481.504,Z 228.513,A -85,B 0,C 180,E1 -6755.654,E2 -6755.654} C_VEL
LIN {X 0,Y 481.464,Z 228.566,A -85,B 0,C 180,E1 -6755.865,E2 -6755.865} C_VEL
LIN {X 0,Y 481.363,Z 234.139,A -85,B 0,C 180,E1 -6758.395,E2 -6758.395} C_VEL
LIN {X 0,Y 481.385,Z 241.999,A -85,B 0,C 180,E1 -6761.992,E2 -6761.992} C_VEL
LIN {X 0,Y 481.296,Z 249.509,A -85,B 0,C 180,E1 -6765.474,E2 -6765.474} C_VEL
LIN {X 0,Y 481.15,Z 256.505,A -85,B 0,C 180,E1 -6768.744,E2 -6768.744} C_VEL
LIN {X 0,Y 481.068,Z 262.225,A -85,B 0,C 180,E1 -6771.422,E2 -6771.422} C_VEL
LIN {X 0,Y 481.014,Z 268.029,A -85,B 0,C 180,E1 -6774.148,E2 -6774.148} C_VEL
LIN {X 0,Y 481.065,Z 270.5,A -85,B 0,C 180,E1 -6775.311,E2 -6775.311} C_VEL
LIN {X 0,Y 482.806,Z 280.961,A -85,B 0,C 180,E1 -6775.702,E2 -6775.702} C_VEL
LIN {X 0,Y 482.611,Z 292.687,A -85,B 0,C 180,E1 -6776.253,E2 -6776.253} C_VEL
LIN {X 0,Y 482.33,Z 302.028,A -85,B 0,C 180,E1 -6776.853,E2 -6776.853} C_VEL
LIN {X 0,Y 482.122,Z 309.949,A -85,B 0,C 180,E1 -6777.49,E2 -6777.49} C_VEL
LIN {X 0,Y 481.933,Z 316.924,A -85,B 0,C 180,E1 -6778.172,E2 -6778.172} C_VEL
LIN {X 0,Y 481.704,Z 323.226,A -85,B 0,C 180,E1 -6778.908,E2 -6778.908} C_VEL
LIN {X 0,Y 481.483,Z 329.271,A -85,B 0,C 180,E1 -6779.754,E2 -6779.754} C_VEL
LIN {X 0,Y 481.285,Z 335.018,A -85,B 0,C 180,E1 -6780.736,E2 -6780.736} C_VEL
LIN {X 0,Y 481.085,Z 341.125,A -85,B 0,C 180,E1 -6782.08,E2 -6782.08} C_VEL
LIN {X 0,Y 480.974,Z 344.743,A -85,B 0,C 180,E1 -6783.165,E2 -6783.165} C_VEL
LIN {X 0,Y 480.915,Z 347.37,A -85,B 0,C 180,E1 -6784.238,E2 -6784.238} C_VEL
LIN {X 0,Y 480.839,Z 348.846,A -85,B 0,C 180,E1 -6785.064,E2 -6785.064} C_VEL
LIN {X 0,Y 480.773,Z 350.087,A -85,B 0,C 180,E1 -6786.486,E2 -6786.486} C_VEL
LIN {X 0,Y 480.753,Z 350.004,A -85,B 0,C 180,E1 -6787.878,E2 -6787.878} C_VEL
LIN {X 0,Y 480.845,Z 348.605,A -85,B 0,C 180,E1 -6789.227,E2 -6789.227} C_VEL
LIN {X 0,Y 480.972,Z 345.832,A -85,B 0,C 180,E1 -6790.551,E2 -6790.551} C_VEL
LIN {X 0,Y 481.049,Z 343.134,A -85,B 0,C 180,E1 -6791.471,E2 -6791.471} C_VEL
LIN {X 0,Y 481.145,Z 340.462,A -85,B 0,C 180,E1 -6792.215,E2 -6792.215} C_VEL
